						// Search next tu for this sequence
						fbSeqGetNextTU(
							Execute:= TRUE, 
							TU_Index:= TU_Index, 
							Destination:= TU_Table[TU_Index].Destination[1], 
							DestinationSlot:= TU_Table[TU_Index].DataSet.DestinationSlot, 
							Sequence:= TU_Table[TU_Index].DataSet.Sequence, 
							SubSequence:= TU_Table[TU_Index].DataSet.SubSequence, 
							Branch := Branch,
							BranchExclusionMode := BranchExclusionMode,
							TU_Table := TU_Table);

						State := 1;
					ELSE
						// Invalid TU data
						Busy := FALSE;
						State := 0;
					END_IF
				ELSE
					// No TU data, not part of a sequence
					Busy := FALSE;
					State := 0;	
				END_IF
			ELSE
				// No TU, stay
				Busy := FALSE;
				State := 0;
			END_IF
		END_IF
	
	// Search Next TU
	1:
		fbSeqGetNextTU(Execute:= FALSE, TU_Table := TU_Table);
		
		IF NOT fbSeqGetNextTU.Busy THEN
			IF NOT fbSeqGetNextTU.Error THEN
				NextTU_Index := fbSeqGetNextTU.NextTU_Index;
				// A next was found, store information to detect TU Data changes
				IF NextTU_Index > 0 THEN			
					M_AddToList(NextTU_Index, TU_Table[NextTU_Index]);
				END_IF
				
				Busy := FALSE;
				State := 0;
			ELSE
				// Error during search
				Error := TRUE;
				Busy := FALSE;
				State := 0;
			END_IF
		END_IF
ELSE
	// Default
	State := 0;
END_CASE

/// Add found data set to list
METHOD PRIVATE M_AddToList : BOOL
VAR_INPUT
	mTU_Index		: DINT;
END_VAR
VAR_IN_OUT
	mTU_Data		: ST_TU_Data;
END_VAR
VAR
	mIdx			: INT;
END_VAR
M_AddToList := FALSE;
		
FOR mIdx := 1 TO MAX_LIST_ENTRIES DO
	/// Check if already a slot is used for that destination
	IF NextTU_List[mIdx].Destination.eFunctionNumber = mTU_Data.Destination[1].eFunctionNumber AND
       NextTU_List[mIdx].Destination.ZoneNumber = mTU_Data.Destination[1].ZoneNumber AND
	   NextTU_List[mIdx].DestinationSlot = mTU_Data.DataSet.DestinationSlot THEN
	   
	    // Replace and store TU Data
	   	NextTU_List[mIdx].TU_Index := mTU_Index;
		NextTU_List[mIdx].Sequence := mTU_Data.DataSet.Sequence;
		NextTU_List[mIdx].SubSequence := mTU_Data.DataSet.SubSequence;
		NextTU_List[mIdx].Destination := mTU_Data.Destination[1];
		NextTU_List[mIdx].DestinationSlot := mTU_Data.DataSet.DestinationSlot;
		NextTU_List[mIdx].TU_ID_HashCode := mTU_Data.TU_ID.HashCode;
		NextTU_List[mIdx].TU_ID := mTU_Data.TU_ID.ASCII;
		NextTU_List[mIdx].AssignmentID := mTU_Data.AssignmentID;
	   	
		M_AddToList := TRUE;
	
	// If an empty slot is found
	ELSIF NextTU_List[mIdx].Destination.eFunctionNumber = E_FunctionNumber.F_BEGIN_FUNCTION THEN
		// Store TU Data
	   	NextTU_List[mIdx].TU_Index := mTU_Index;
		NextTU_List[mIdx].Sequence := mTU_Data.DataSet.Sequence;
		NextTU_List[mIdx].SubSequence := mTU_Data.DataSet.SubSequence;
		NextTU_List[mIdx].Destination := mTU_Data.Destination[1];
		NextTU_List[mIdx].DestinationSlot := mTU_Data.DataSet.DestinationSlot;
		NextTU_List[mIdx].TU_ID_HashCode := mTU_Data.TU_ID.HashCode;
		NextTU_List[mIdx].TU_ID := mTU_Data.TU_ID.ASCII;
		NextTU_List[mIdx].AssignmentID := mTU_Data.AssignmentID;
		
		M_AddToList := TRUE;
		
		ListCount := ListCount + 1;
	END_IF	
END_FOR
END_METHOD

/// Clears next TU list.
/// Returns true if succesful.
METHOD M_ClearList : BOOL
M_ClearList := MEMSET(ADR(NextTU_List), 0, SIZEOF(NextTU_List)) > 0;
END_METHOD

/// Checks if requesting TU is next in sequence
METHOD M_IsNextInSequence : BOOL // True = Next in Sequence, otherwise FALSE
VAR_INPUT
	mTU_Index		: DINT; // Requesting TU Index
END_VAR
VAR_IN_OUT
	mTU_Data		: ST_TU_Data; // Tu Data
END_VAR
VAR
	mIdx			: INT; // Iterator
END_VAR
M_IsNextInSequence := FALSE;
		
FOR mIdx := 1 TO ListCount DO
	// Check if an index is recorded as next
	IF mTU_Index = NextTU_List[mIdx].TU_Index THEN
		/// Ensure that recorded tu data entry is still the same as requesting Tu data
		IF mTU_Data.DataSet.Sequence = NextTU_List[mIdx].Sequence AND
		   mTU_Data.DataSet.SubSequence = NextTU_List[mIdx].SubSequence AND
		   mTU_Data.TU_ID.ASCII = NextTU_List[mIdx].TU_ID AND
		   mTU_Data.Destination[1].eFunctionNumber = NextTU_List[mIdx].Destination.eFunctionNumber AND
		   mTU_Data.Destination[1].ZoneNumber = NextTU_List[mIdx].Destination.ZoneNumber AND 
		   mTU_Data.DataSet.DestinationSlot = NextTU_List[mIdx].DestinationSlot THEN
		   
			M_IsNextInSequence := TRUE;
			RETURN;
		END_IF	
	END_IF
END_FOR
END_METHOD

END_FUNCTION_BLOCK

// ---- 20_Product/30_Toolbox/16_Sequencing/11_Strategies/FB_SeqEstimateNextTU.TcPOU
/// Estimates next awaiting TU after the requesting one of one specific destination.
FUNCTION_BLOCK FB_SeqEstimateNextTU IMPLEMENTS I_SeqEstimateNext
(************************************************************************************** 
* 	Application 		: BoxControl Framework 
* 	Revision 			: $Revision: 404877 $ 
* 	Revision date 		: $Date: 2018-04-26 14:10:34 +0200 (Thu, 26 Apr 2018) $ 
* 	Last changed by 	: $Author: b7ernsb $ 
* 	URL 				: $URL: http://almscdc.swisslog.com/repo/SWPD/Development/BoxControlFramework/21_Projects/BCF_2.0/trunk/BCF/BCF/JumpStart/20_Product/10_App/12_E_Functions/10_Lib/10_Conv/FB_FunctionConv.TcPOU $ 
* ------------------------------------------------------------------------------------ 
* 	© Swisslog AG 
* 	Swisslog is not liable for any usage of this source code that is not agreed 
* 	on between Swisslog and the other party. The mandatory legal liability remains 
* 	unaffected. 
* ------------------------------------------------------------------------------------ 
* 	Revision History: 
* 
* 	VERSION 		DATE 			INITIALS 			DESCRIPTION 
* 	0.1 			23.05.2018 		mbo 				Created.
*	0.2				31.10.2018		mbo					Race condition fixed for NextTUIndex
* 
**************************************************************************************)
VAR_INPUT
	Execute					: BOOL; // Requires rising edge for new request
	TU_Present				: BOOL; // A TU is present on branch A
	TU_Index				: DINT; // Waiting TU data index A
	Destination				: ST_PositionIdent; // Estimates next TU for this destination
	DestinationSlot			: INT; // Estimates next TU for this destination slot
	Branch					: I_BranchCheckpoint; // Branch to check for next branch
	BranchExclusionMode		: BOOL := FALSE; // False = TU on a branch is possible next, TRUE = TU on a branch is excluded as possible next
END_VAR
VAR_OUTPUT
	Busy					: BOOL; // Process ongoing
	Error					: BOOL; // Error during process (configuration error)
	NextTU_Index			: DINT; // Next expected TU of this sequence
END_VAR
VAR_IN_OUT
	TU_Table				: ARRAY[0..Conveyor.NUMBER_OF_TU_DATA] OF ST_TU_Data; // TU Table
END_VAR
VAR
	State					: INT; // State machine 0: Request 1: Search
	fbTrigExecute			: R_TRIG; // Trigger new request
	TU_DataChanged			: BOOL; // Data of stored NextTU have changed
	TU_LocationChanged		: BOOL; // Location of stored NextTU has changed
	TU_IsPartOfDestSequence : BOOL; // TU is part of the sequence to this destination
	SequenceDataPresent 	: BOOL; // Sequence data available
	NextAssignmentID		: UDINT; // Stored next assignment ID
	NextDestination			: ST_PositionIdent; // Stored destination information
	NextDestinationSlot		: INT; // Stored destination slot
	NextTU_ID				: STRING(Conveyor.TU_ID_STRINGLENGTH); // Stored next TU-ID HashCode
	NextSequence			: ULINT; // Stored next sequence
	NextSubSequence			: DINT; // Stored next sub sequence
	NextCheckpointID		: STRING(5); // Stored next checkpoint ID
	NextHaltSequencing		: BOOL; // Stored next halt sequencing bit
	fbSeqGetNextTU			: FB_SeqGetNextTU; // Get next following TU of this sequence
END_VAR

// Monitor new request trigger
fbTrigExecute(CLK := Execute);

CASE State OF
	// Wait for a new TU
	0:
		// Wait for new start trigger
		IF fbTrigExecute.Q THEN
			// Validate inputs
			IF Branch = 0 THEN
				Error := TRUE;
				RETURN;
			END_IF
			
			// Process started...
			Busy := TRUE;
			Error := FALSE;

			// When a requesting TU is present
			IF TU_Present THEN
				// If already a next TU was determined on a previous search, 
				// check if state or position has changed of it
				IF NextTU_Index > 0 THEN
					// Detect if the data of the monitored TU index has changed (e.g. TU data Add/Remove/Update)		
					TU_DataChanged := TU_Table[NextTU_Index].AssignmentID <> NextAssignmentID OR
									  TU_Table[NextTU_Index].TU_ID.ASCII <> NextTU_ID OR
									  TU_Table[NextTU_Index].DataSet.Sequence <> NextSequence OR
									  TU_Table[NextTU_Index].DataSet.SubSequence <> NextSubSequence OR
                                      TU_Table[NextTU_Index].Destination[1].eFunctionNumber <> NextDestination.eFunctionNumber OR
  									  TU_Table[NextTU_Index].Destination[1].ZoneNumber <> NextDestination.ZoneNumber OR
									  TU_Table[NextTU_Index].DataSet.DestinationSlot <> NextDestinationSlot OR
									  TU_Table[NextTU_Index].DataSet.HaltSequencing <> NextHaltSequencing;
			
					// Detect if the TU has changed the location (e.g. entered a new path)
					TU_LocationChanged := TU_Table[NextTU_Index].DataSet.CheckpointID <> NextCheckpointID;

					// Data changed, new release request		  
					IF TU_DataChanged OR TU_LocationChanged THEN
						M_ClearNextTU_Data();
					END_IF
				END_IF
					
				IF NextTU_Index > 0 THEN
					// No change of expected TU
					Busy := FALSE;
					State := 0;
				ELSIF TU_Index > 0 THEN
					// If the TU consists of sequencing information
					SequenceDataPresent := TU_Table[TU_Index].DataSet.Sequence > 0 AND
					                       TU_Table[TU_Index].Destination[1].eFunctionNumber > 0;
										   
					TU_IsPartOfDestSequence := TU_Table[TU_Index].Destination[1].eFunctionNumber = Destination.eFunctionNumber AND
					 						   TU_Table[TU_Index].Destination[1].ZoneNumber = Destination.ZoneNumber AND
											   TU_Table[TU_Index].DataSet.DestinationSlot = DestinationSlot;
					
					IF SequenceDataPresent AND TU_IsPartOfDestSequence THEN
						fbSeqGetNextTU(
							Execute:= TRUE, 
							TU_Index:= TU_Index, 
							Destination:= TU_Table[TU_Index].Destination[1], 
							DestinationSlot:= TU_Table[TU_Index].DataSet.DestinationSlot, 
							Sequence:= TU_Table[TU_Index].DataSet.Sequence, 
							SubSequence:= TU_Table[TU_Index].DataSet.SubSequence, 
							Branch := Branch,
							BranchExclusionMode := BranchExclusionMode,
							TU_Table := TU_Table);
							
						State := 1;
					ELSE
						// Invalid TU data
						Busy := FALSE;
						State := 0;
					END_IF
				ELSE
					// No TU data, not part of a sequence
					Busy := FALSE;
					State := 0;	
				END_IF
			ELSE
				// No TU, stay
				Busy := FALSE;
				State := 0;
			END_IF
		END_IF
	
	// Search Next TU
	1:
		fbSeqGetNextTU(
			Execute:= FALSE, 
			TU_Index:= TU_Index, 
			Destination:= TU_Table[TU_Index].Destination[1], 
			DestinationSlot:= TU_Table[TU_Index].DataSet.DestinationSlot, 
			Sequence:= TU_Table[TU_Index].DataSet.Sequence, 
			SubSequence:= TU_Table[TU_Index].DataSet.SubSequence, 
			Branch := Branch,
			BranchExclusionMode := BranchExclusionMode,
			NextTU_Index => NextTU_Index,
			TU_Table := TU_Table);
		
		IF NOT fbSeqGetNextTU.Busy THEN
			IF NOT fbSeqGetNextTU.Error THEN
				// A next was found, store information to detect TU Data changes
				IF NextTU_Index > 0 THEN
					NextAssignmentID := TU_Table[NextTU_Index].AssignmentID; 
					NextTU_ID := TU_Table[NextTU_Index].TU_ID.ASCII;
					NextSequence := TU_Table[NextTU_Index].DataSet.Sequence;
					NextSubSequence	:= TU_Table[NextTU_Index].DataSet.SubSequence;
					NextCheckpointID := TU_Table[NextTU_Index].DataSet.CheckpointID;
					NextDestination := TU_Table[NextTU_Index].Destination[1];
					NextDestinationSlot := TU_Table[NextTU_Index].DataSet.DestinationSlot;
					NextHaltSequencing := TU_Table[NextTU_Index].DataSet.HaltSequencing;

				// No next found for this specific destination
				ELSE
					M_ClearNextTU_Data();
				END_IF
				
				Busy := FALSE;
				State := 0;
			ELSE
				// Error during search
				Error := TRUE;
				Busy := FALSE;
				State := 0;
			END_IF
		END_IF
ELSE
	// Default
	State := 0;
END_CASE

/// Reset next expected TU, so on a new request a new search is triggered
METHOD M_ResetExpectedTU 
VAR_INPUT
END_VAR
NextTU_Index := 0;
END_METHOD

/// Clears next tu data
METHOD PROTECTED M_ClearNextTU_Data
VAR_INPUT
END_VAR
NextTU_Index := 0;
NextAssignmentID := 0; 
NextTU_ID := '';
NextSequence := 0;
NextSubSequence	:= 0;
NextCheckpointID := '';
NextDestination.eFunctionNumber := 0;
NextDestination.ZoneNumber := 0;
NextDestinationSlot := 0;
NextHaltSequencing :=  FALSE;
END_METHOD

/// Checks if requesting TU is next in sequence
METHOD M_IsNextInSequence : BOOL // True = Next in Sequence, otherwise FALSE
VAR_INPUT
	mTU_Index		: DINT; // Requesting TU Index
END_VAR
VAR_IN_OUT
	mTU_Data			: ST_TU_Data; // Tu Data
END_VAR

IF NextTU_Index > 0 THEN
	// Check whether the requesting TU is the same, as the next sequence TU was stored
	IF TU_Index = NextTU_Index AND
	   mTU_Data.DataSet.Sequence = NextSequence AND
	   mTU_Data.DataSet.SubSequence = NextSubSequence AND
	   mTU_Data.TU_ID.ASCII = NextTU_ID AND
	   mTU_Data.DataSet.CheckpointID = NextCheckpointID AND
	   mTU_Data.Destination[1].eFunctionNumber = NextDestination.eFunctionNumber AND
	   mTU_Data.Destination[1].ZoneNumber = NextDestination.ZoneNumber AND 
	   mTU_Data.DataSet.DestinationSlot = NextDestinationSlot THEN
	   
	   	// Release
		M_IsNextInSequence := TRUE;
	ELSE
	   M_IsNextInSequence := FALSE;
	END_IF
ELSE
	M_IsNextInSequence := FALSE;
END_IF
END_METHOD

END_FUNCTION_BLOCK

// ---- 20_Product/30_Toolbox/16_Sequencing/11_Strategies/FB_SeqEstimateStreamRange.TcPOU
/// Estimates all next awaiting TUs of one specific destination stream considering 
/// the configured branch.
FUNCTION_BLOCK FB_SeqEstimateStreamRange 
(************************************************************************************** 
* 	Application 		: BoxControl Framework 
* 	Revision 			: $Revision: 404877 $ 
* 	Revision date 		: $Date: 2018-04-26 14:10:34 +0200 (Thu, 26 Apr 2018) $ 
* 	Last changed by 	: $Author: b7ernsb $ 
* 	URL 				: $URL: http://almscdc.swisslog.com/repo/SWPD/Development/BoxControlFramework/21_Projects/BCF_2.0/trunk/BCF/BCF/JumpStart/20_Product/10_App/12_E_Functions/10_Lib/10_Conv/FB_FunctionConv.TcPOU $ 
* ------------------------------------------------------------------------------------ 
* 	© Swisslog AG 
* 	Swisslog is not liable for any usage of this source code that is not agreed 
* 	on between Swisslog and the other party. The mandatory legal liability remains 
* 	unaffected. 
* ------------------------------------------------------------------------------------ 
* 	Revision History: 
* 
* 	VERSION 		DATE 			INITIALS 			DESCRIPTION 
* 	0.1 			23.05.2018 		mbo 				Created.
*	0.2				08.02.2019		mbo					Renamed + Racecondition
* 
**************************************************************************************)
VAR_INPUT
	Execute					: BOOL; // Requires rising edge for new request
	TU_Present				: BOOL; // A TU is present on branch A
	TU_Index				: DINT; // Waiting TU data index A
	Destination				: ST_PositionIdent; // Estimates next TU for this destination
	DestinationSlot			: INT; // Estimates next TU for this destination slot
	Branch					: I_BranchCheckpoint; // Branch to check for next branch
	BranchExclusionMode		: BOOL := FALSE; // False = TU on a branch is possible next, TRUE = TU on a branch is excluded as possible next
	RangeLimit				: INT; // Specifies how many entries of the list serve as valid. (0=All available)
END_VAR
VAR_OUTPUT
	Busy					: BOOL; // Process ongoing
	Error					: BOOL; // Error during process (configuration error)
	NextTU_Index			: DINT; // Next expected TU of this sequence
END_VAR
VAR_IN_OUT
	TU_Table				: ARRAY[0..Conveyor.NUMBER_OF_TU_DATA] OF ST_TU_Data; // TU Table
END_VAR
VAR
	State					: INT; // State machine 0: Request 1: Search
	fbTrigExecute			: R_TRIG; // Trigger new request
	TU_DataChanged			: BOOL; // Data of stored NextTU have changed
	TU_LocationChanged		: BOOL; // Location of stored NextTU has changed
	TU_IsPartOfDestSequence : BOOL; // TU is part of the sequence to this destination
	SequenceDataPresent 	: BOOL; // Sequence data available
	NextAssignmentID		: UDINT; // Stored next assignment ID
	NextDestination			: ST_PositionIdent; // Stored destination information
	NextDestinationSlot		: INT; // Stored destination slot
	NextTU_ID				: STRING(Conveyor.TU_ID_STRINGLENGTH); // Stored next TU-ID HashCode
	NextSequence			: ULINT; // Stored next sequence
	NextSubSequence			: DINT; // Stored next sub sequence
	NextCheckpointID		: STRING(5); // Stored next checkpoint ID
	NextHaltSequencing		: BOOL; // Stored next halt sequencing bit
	fbSeqBuildStream		: FB_SeqBuildStream; // Instance to build range of stream
END_VAR

// Monitor new request trigger
fbTrigExecute(CLK := Execute);

CASE State OF
	// Wait for a new TU
	0:
		// Wait for new start trigger
		IF fbTrigExecute.Q THEN
			// Validate inputs
			IF Branch = 0 THEN
				Error := TRUE;
				RETURN;
			END_IF
			
			// Process started...
			Busy := TRUE;
			Error := FALSE;

			// When a requesting TU is present
			IF TU_Present THEN
				// If already a next TU was determined on a previous search, 
				// check if state or position has changed of it
				IF NextTU_Index > 0 THEN
					// Detect if the data of the monitored TU index has changed (e.g. TU data Add/Remove/Update)		
					TU_DataChanged := TU_Table[NextTU_Index].AssignmentID <> NextAssignmentID OR
									  TU_Table[NextTU_Index].TU_ID.ASCII <> NextTU_ID OR
									  TU_Table[NextTU_Index].DataSet.Sequence <> NextSequence OR
									  TU_Table[NextTU_Index].DataSet.SubSequence <> NextSubSequence OR
                                      TU_Table[NextTU_Index].Destination[1].eFunctionNumber <> NextDestination.eFunctionNumber OR
  									  TU_Table[NextTU_Index].Destination[1].ZoneNumber <> NextDestination.ZoneNumber OR
									  TU_Table[NextTU_Index].DataSet.DestinationSlot <> NextDestinationSlot OR
									  TU_Table[NextTU_Index].DataSet.HaltSequencing <> NextHaltSequencing;
			
					// Detect if the TU has changed the location (e.g. entered a new path)
					TU_LocationChanged := TU_Table[NextTU_Index].DataSet.CheckpointID <> NextCheckpointID;

					// Data changed, new release request		  
					IF TU_DataChanged OR TU_LocationChanged THEN
						M_ClearNextTU_Data();
					END_IF
				END_IF
					
				IF NextTU_Index > 0 THEN
					// No change of expected TU
					Busy := FALSE;
					State := 0;
				ELSIF TU_Index > 0 THEN
					// If the TU consists of sequencing information
					SequenceDataPresent := TU_Table[TU_Index].DataSet.Sequence > 0 AND
					                       TU_Table[TU_Index].Destination[1].eFunctionNumber > 0;
										   
					TU_IsPartOfDestSequence := TU_Table[TU_Index].Destination[1].eFunctionNumber = Destination.eFunctionNumber AND
					 						   TU_Table[TU_Index].Destination[1].ZoneNumber = Destination.ZoneNumber AND
											   TU_Table[TU_Index].DataSet.DestinationSlot = DestinationSlot;
					
					IF SequenceDataPresent AND TU_IsPartOfDestSequence THEN
						
						fbSeqBuildStream(
							Execute:= TRUE,
							Destination:= TU_Table[TU_Index].Destination[1], 
							DestinationSlot:= TU_Table[TU_Index].DataSet.DestinationSlot, 
							Branch := Branch,
							BranchExclusionMode := BranchExclusionMode,
							TU_Table := TU_Table);
							
						State := 1;
					ELSE
						// Invalid TU data
						Busy := FALSE;
						State := 0;
					END_IF
				ELSE
					// No TU data, not part of a sequence
					Busy := FALSE;
					State := 0;	
				END_IF
			ELSE
				// No TU, stay
				Busy := FALSE;
				State := 0;
			END_IF
		END_IF
	
	// Search Next TU
	1:
		fbSeqBuildStream(
			Execute:= FALSE,
			Destination:= TU_Table[TU_Index].Destination[1], 
			DestinationSlot:= TU_Table[TU_Index].DataSet.DestinationSlot, 
			Branch := Branch,
			BranchExclusionMode := BranchExclusionMode,
			NextTU_Index => NextTU_Index,
			TU_Table := TU_Table);
		
		IF NOT fbSeqBuildStream.Busy THEN
			IF NOT fbSeqBuildStream.Error THEN
				// A next was found, store information to detect TU Data changes
				IF NextTU_Index > 0 THEN
					NextAssignmentID := TU_Table[NextTU_Index].AssignmentID; 
					NextTU_ID := TU_Table[NextTU_Index].TU_ID.ASCII;
					NextSequence := TU_Table[NextTU_Index].DataSet.Sequence;
					NextSubSequence	:= TU_Table[NextTU_Index].DataSet.SubSequence;
					NextCheckpointID := TU_Table[NextTU_Index].DataSet.CheckpointID;
					NextDestination := TU_Table[NextTU_Index].Destination[1];
					NextDestinationSlot := TU_Table[NextTU_Index].DataSet.DestinationSlot;
					NextHaltSequencing := TU_Table[NextTU_Index].DataSet.HaltSequencing;
					
				// No next found for this specific destination
				ELSE
					M_ClearNextTU_Data();
				END_IF
				
				Busy := FALSE;
				State := 0;
			ELSE
				// Error during search
				Error := TRUE;
				Busy := FALSE;
				State := 0;
			END_IF
		END_IF
ELSE
	// Default
	State := 0;
END_CASE

/// Reset next expected TU, so on a new request a new search is triggered
METHOD M_ResetExpectedTU 
VAR_INPUT
END_VAR
NextTU_Index := 0;
END_METHOD

/// Checks if requesting TU is next in sequence
METHOD M_IsNextInSequence : BOOL // True = Next in Sequence, otherwise FALSE
VAR_INPUT
	mTU_Index		: DINT; // Requesting TU Index
END_VAR
VAR_IN_OUT
	mTU_Data			: ST_TU_Data; // Tu Data
END_VAR

IF NextTU_Index > 0 THEN
	M_IsNextInSequence := fbSeqBuildStream.M_IsTU_OnStream(
												mRangeLimit := RangeLimit,
												mTU_Index := TU_Index,
												mTU_Data := mTU_Data);
ELSE
	M_IsNextInSequence := FALSE;
END_IF
END_METHOD

/// Clears next tu data
METHOD PROTECTED M_ClearNextTU_Data
VAR_INPUT
END_VAR
NextTU_Index := 0;
NextAssignmentID := 0; 
NextTU_ID := '';
NextSequence := 0;
NextSubSequence	:= 0;
NextCheckpointID := '';
NextDestination.eFunctionNumber := 0;
NextDestination.ZoneNumber := 0;
NextDestinationSlot := 0;
END_METHOD

END_FUNCTION_BLOCK

// ---- 20_Product/30_Toolbox/16_Sequencing/11_Strategies/FB_SeqMerge2W.TcPOU
/// Sequence strategy Merge 2-Way
/// This strategy is able to ensure sequencing from two branches.
/// Remark: Decision can take multiple cycles, check busy and reset FB before new request.
/// Uses recursive calls - User has to ensure to not generate a loop (Tested up to 350 jumps)
FUNCTION_BLOCK FB_SeqMerge2W IMPLEMENTS I_BranchCheckpoint
(************************************************************************************** 
* 	Application 		: BoxControl Framework 
* 	Revision 			: $Revision: 404877 $ 
* 	Revision date 		: $Date: 2018-04-26 14:10:34 +0200 (Thu, 26 Apr 2018) $ 
* 	Last changed by 	: $Author: b7ernsb $ 
* 	URL 				: $URL: http://almscdc.swisslog.com/repo/SWPD/Development/BoxControlFramework/21_Projects/BCF_2.0/trunk/BCF/BCF/JumpStart/20_Product/10_App/12_E_Functions/10_Lib/10_Conv/FB_FunctionConv.TcPOU $ 
* ------------------------------------------------------------------------------------ 
* 	© Swisslog AG 
* 	Swisslog is not liable for any usage of this source code that is not agreed 
* 	on between Swisslog and the other party. The mandatory legal liability remains 
* 	unaffected. 
* ------------------------------------------------------------------------------------ 
* 	Revision History: 
* 
* 	VERSION 		DATE 			INITIALS 			DESCRIPTION 
* 	0.1 			01.05.2018 		mbo 				Created.
* 
**************************************************************************************)
VAR_INPUT
	Execute					: BOOL; // Requires rising edge for new request
	CheckpointID			: STRING(5); // Checkpoint ID, used to identify location of TUs
	TU_PresentA				: BOOL; // A TU is present on branch A
	TU_IndexA				: DINT; // Waiting TU data index A
	TU_PresentB 			: BOOL; // A TU is present on branch B
	TU_IndexB				: DINT; // Waiting TU data index B
	iBranchA				: I_BranchCheckpoint; // Previous decision point on this branch
	iBranchB				: I_BranchCheckpoint; // Previous decision point on this branch
	iEstimateNextServiceA	: I_SeqEstimateNext; // Service to estimate possible next in order to save calculation time (optional)
	iEstimateNextServiceB	: I_SeqEstimateNext; // Service to estimate possible next in order to save calculation time (optional)
	EnableWarningA			: BOOL; // When enabled, warning is active if a TU is waiting, RisingEdge restarts Timer
	EnableWarningB			: BOOL; // When enabled, warning is active if a TU is waiting, RisingEdge restarts Timer
END_VAR

VAR_IN_OUT 
	TU_Table				: ARRAY[0..Conveyor.NUMBER_OF_TU_DATA] OF ST_TU_Data; // TU Table
END_VAR

VAR_OUTPUT
	Busy					: BOOL; // Process ongoing
	Error					: BOOL; // Error during process
	ReleaseA				: BOOL; // Release TU on branch A
	ReleaseB				: BOOL; // Release TU on branch B
	TimeoutWaitA			: BOOL; // Warning, TU is waiting longer than P_WarningTime
	TimeoutWaitB			: BOOL; // Warning, TU is waiting longer than P_WarningTime
END_VAR

VAR
	fbBranchA				: FB_SeqBranch; // Branch A 
	fbBranchB				: FB_SeqBranch; // Branch B
	UpdateCheckpointID		: BOOL; // Enable update ceckpoint IDs of waiting Tus
	WarningTime				: TIME := SequencingParameter.DEFAULT_WARNING_TIME; // Time after a warning gets reported.
	fbWarnA					: TON; // Timer warning A
	fbWarnB					: TON; // Timer warning B
END_VAR

// Check inputs
IF TU_IndexA < 0 OR TU_IndexB < 0 THEN
	Error := TRUE;
	RETURN;
END_IF

// Initialize values
Error := FALSE;

// If branch A is configured, update waiting TU with Checkpoint ID
IF iBranchA <> 0 AND UpdateCheckpointID THEN
	F_UpdateCheckpointID(
		Enable := TU_PresentA AND TU_IndexA > 0,
		CheckpointID := iBranchA.P_CheckpointID,
		TU_Data := TU_Table[TU_IndexA]);
END_IF

// If branch B is configured, update waiting TU with Checkpoint ID
IF iBranchB <> 0 AND UpdateCheckpointID THEN
	F_UpdateCheckpointID(
		Enable := TU_PresentB AND TU_IndexB > 0,
		CheckpointID := iBranchB.P_CheckpointID,
		TU_Data := TU_Table[TU_IndexB]);	
END_IF

fbBranchA(
	Execute:= Execute, 
	TU_Present:= TU_PresentA, 
	TU_Index:= TU_IndexA, 
	Branch:= iBranchA, 
	iEstimateNextService:= iEstimateNextServiceA, 
	Release=> ReleaseA, 
	TU_Table:= TU_Table);
	
fbBranchB(
	Execute:= Execute, 
	TU_Present:= TU_PresentB, 
	TU_Index:= TU_IndexB, 
	Branch:= iBranchB, 
	iEstimateNextService:= iEstimateNextServiceB, 
	Release=> ReleaseB, 
	TU_Table:= TU_Table);
	
Busy := fbBranchA.Busy OR fbBranchB.Busy;
Error := fbBranchA.Error OR fbBranchB.Error;

fbWarnA(IN := EnableWarningA AND TU_PresentA, PT := WarningTime);
fbWarnB(IN := EnableWarningB AND TU_PresentB, PT := WarningTime);

TimeoutWaitA := fbWarnA.Q;
TimeoutWaitB := fbWarnB.Q;

/// Searches if a checkpoint can be found on a specific branch
/// Returns true if found, false = not found
METHOD M_IsOnBranches : BOOL
VAR_INPUT
	mRecursive	: BOOL := FALSE; // Search recursive through the whole tree
END_VAR
VAR_IN_OUT CONSTANT
	// Last checkpoint id	
	mCheckpointID	: STRING(5);
END_VAR

IF mCheckpointID = '' THEN
	M_IsOnBranches := FALSE;
	RETURN;
END_IF

IF mCheckpointID = P_CheckpointID THEN
	M_IsOnBranches := TRUE;
	RETURN;
END_IF

// When its requested that its branches are checked as well
IF mRecursive THEN
	IF iBranchA <> 0 THEN
		 IF iBranchA.M_IsOnBranches(TRUE, mCheckpointId) THEN;
			M_IsOnBranches := TRUE;
			RETURN;
		END_IF
	END_IF
	
	IF iBranchB <> 0 THEN
		IF iBranchB.M_IsOnBranches(TRUE, mCheckpointId) THEN;
			M_IsOnBranches := TRUE;
			RETURN;
		END_IF
	END_IF
END_IF
END_METHOD

METHOD M_Reset : BOOL
VAR_INPUT
END_VAR
fbBranchA.M_Reset();
fbBranchB.M_Reset();
END_METHOD

/// Identifier for checkpoint
{attribute 'monitoring' := 'call'}
{attribute 'suppress_wrn_C0410'}
PROPERTY P_CheckpointID : REFERENCE TO STRING(5)
GET
P_CheckpointID REF= CheckpointID;
END_GET
END_PROPERTY

/// TU Entries scanned per cycle
PROPERTY P_EntriesPerCycle : DINT // Default 600
GET
P_EntriesPerCycle := fbBranchA.P_EntriesPerCycle;
END_GET
SET
fbBranchA.P_EntriesPerCycle := P_EntriesPerCycle;
fbBranchB.P_EntriesPerCycle := P_EntriesPerCycle;
END_SET
END_PROPERTY

/// When enabled, Checkpoint ID of waiting TUs is updated automatically with previous Branch ID
PROPERTY P_UpdateCheckpointID : BOOL
GET
P_UpdateCheckpointID := UpdateCheckpointID;
END_GET
SET
UpdateCheckpointID := P_UpdateCheckpointID;
END_SET
END_PROPERTY

/// Time after Warning gets reported
PROPERTY P_WarningTime : TIME
GET
P_WarningTime := WarningTime;
END_GET
SET
WarningTime := P_WarningTime;
END_SET
END_PROPERTY

END_FUNCTION_BLOCK

// ---- 20_Product/30_Toolbox/16_Sequencing/12_Helper/FB_SeqConveyorLane.TcPOU
// Object representing a conveyor lane consisting of multiple zones
FUNCTION_BLOCK FB_SeqConveyorLane
(************************************************************************************** 
* 	Application 		: BoxControl Framework 
* 	Revision 			: $Revision: 404877 $ 
* 	Revision date 		: $Date: 2018-04-26 14:10:34 +0200 (Thu, 26 Apr 2018) $ 
* 	Last changed by 	: $Author: b7ernsb $ 
* 	URL 				: $URL: http://almscdc.swisslog.com/repo/SWPD/Development/BoxControlFramework/21_Projects/BCF_2.0/trunk/BCF/BCF/JumpStart/20_Product/10_App/12_E_Functions/10_Lib/10_Conv/FB_FunctionConv.TcPOU $ 
* ------------------------------------------------------------------------------------ 
* 	© Swisslog AG 
* 	Swisslog is not liable for any usage of this source code that is not agreed 
* 	on between Swisslog and the other party. The mandatory legal liability remains 
* 	unaffected. 
* ------------------------------------------------------------------------------------ 
* 	Revision History: 
* 
* 	VERSION 		DATE 			INITIALS 			DESCRIPTION 
* 	0.1 			06.05.2019 		ber 				Created.

* 
**************************************************************************************)
VAR_INPUT
	Positions						: ARRAY [1..MAX_LANE_SIZE] OF ST_PositionIdent; // Index 1: Outfeed position of the lane 
END_VAR
VAR
	PositionCount					: DINT; // Amount of positions in the lane
	OnlySequencingTU				: BOOL:= TRUE; // Only allow TU with sequencing data to enter the lane
	Idx								: DINT;
END_VAR

VAR CONSTANT
	MAX_LANE_SIZE					: DINT:=SequencingParameter.MAX_LANE_SIZE; // Maximal number of zones in a conveyor lane
END_VAR

PositionCount:= 0;	
// Determine amount of positions in the lane
FOR Idx:=1 TO MAX_LANE_SIZE DO
	IF Positions[Idx].eFunctionNumber>0 THEN
		PositionCount:= PositionCount+1;
	END_IF
END_FOR

/// Returns all TU indices currently present in the lane
METHOD M_GetAllTU : BOOL // True = execution sucessfull, else false
VAR_IN_OUT
	mTU_Indices	: ARRAY [*] OF DINT; // List of all TU data indices in the lane
END_VAR
VAR
	mIdx		: DINT;
	mTU_Index	: DINT;
	mCount		: DINT;
END_VAR
MEMSET(ADR(mTU_Indices^), 0,  DINT_TO_UDINT((UPPER_BOUND(mTU_Indices,1)- LOWER_BOUND(mTU_Indices,1)+1)*SIZEOF(mTU_Indices^)));	
mCount:= LOWER_BOUND(mTU_Indices,1);
M_GetAllTU:= TRUE;	

// Loop through lane
FOR mIdx:=1 TO PositionCount DO	
	
	mTU_Index:= F_GetTU_DataIndex(Positions[mIdx].eFunctionNumber, Positions[mIdx].ZoneNumber);
	
	// If a TU index is present on the zone	
	IF mTU_Index > 0 THEN

		// Input array has enough space
		IF mCount <= UPPER_BOUND( mTU_Indices,1) THEN
			
			mTU_Indices[mCount]:= mTU_Index;
			mCount:= mCount+1;
		
		ELSE // Input array too small
	
			MEMSET(ADR(mTU_Indices^), 0, DINT_TO_UDINT((UPPER_BOUND(mTU_Indices,1)- LOWER_BOUND(mTU_Indices,1)+1)*SIZEOF(mTU_Indices^)));		
			M_GetAllTU:= FALSE;	
			EXIT;		
		END_IF

	END_IF
END_FOR
END_METHOD

// Get TU Index on first occupied position (nearest to the infeed)
METHOD M_GetFirstTU : DINT // TU index
VAR
	mIdx				: DINT;
END_VAR
VAR_INST
	TransportCtrlData	: ST_TransportControlData;	
END_VAR
M_GetFirstTU:=0;

// Loop through lane from infeed to outfeed
FOR mIdx:=0 TO PositionCount-1 DO	
	
	TransportCtrlData:= F_GetTransportControlData(Positions[PositionCount-mIdx].eFunctionNumber, Positions[PositionCount-mIdx].ZoneNumber);

	// Finish search when a TU was found	
	IF  TransportCtrlData.NumberOfPresentTUs > 0 THEN
		M_GetFirstTU:=F_GetTU_DataIndex( Positions[PositionCount-mIdx].eFunctionNumber, Positions[PositionCount-mIdx].ZoneNumber);
		EXIT;
	END_IF
	
END_FOR
END_METHOD

// Get TU Index on last occupied position (nearest to the outfeed)
METHOD M_GetLastTU : DINT // TU index
VAR
	mIdx				: DINT;
END_VAR
VAR_INST
	TransportCtrlData	: ST_TransportControlData;	
END_VAR
M_GetLastTU:=0;

// Loop through lane from outfeed to infeed
FOR mIdx:=1 TO PositionCount DO	
	
	TransportCtrlData:= F_GetTransportControlData(Positions[mIdx].eFunctionNumber, Positions[mIdx].ZoneNumber);
	
	// Finish search when a TU was found
	IF  TransportCtrlData.NumberOfPresentTUs > 0 THEN
		M_GetLastTU:= F_GetTU_DataIndex( Positions[mIdx].eFunctionNumber, Positions[mIdx].ZoneNumber);
		EXIT;
	END_IF
	
END_FOR
END_METHOD

// Returns number of empty zones in the lane
METHOD M_GetNrOfEmptyZones : DINT 
VAR
	mIdx				: DINT;
	mEmptyPosition_Count: DINT;
END_VAR
VAR_INST
	TransportCtrlData	: ST_TransportControlData;	
END_VAR
// Loop through lane from outfeed to infeed
FOR mIdx:=1 TO PositionCount DO	
	
	TransportCtrlData:= F_GetTransportControlData(Positions[mIdx].eFunctionNumber, Positions[mIdx].ZoneNumber);
	
	// Increase count when no TU is present on the zone
	IF  TransportCtrlData.NumberOfPresentTUs = 0 THEN
		mEmptyPosition_Count:=mEmptyPosition_Count+1;
	END_IF
	
END_FOR

M_GetNrOfEmptyZones:= mEmptyPosition_Count;
END_METHOD

// Returns number of occupied zones in the lane
METHOD M_GetNrOfOccupiedZones : DINT 
VAR
	mIdx				: DINT;
	mTU_Count			: DINT;
END_VAR
VAR_INST
	TransportCtrlData	: ST_TransportControlData;	
END_VAR
// Loop through lane from outfeed to infeed
FOR mIdx:=1 TO PositionCount DO	
	
	TransportCtrlData:= F_GetTransportControlData(Positions[mIdx].eFunctionNumber, Positions[mIdx].ZoneNumber);

	// Increase count when TU is present on the zone	
	IF  TransportCtrlData.NumberOfPresentTUs > 0 THEN
		mTU_Count:=mTU_Count+1;
	END_IF
	
END_FOR

M_GetNrOfOccupiedZones:= mTU_Count;
END_METHOD

/// Returns all TU indices (which have sequencing data)  after the last sequence error (sequence error nearest to the lane outfeed)
METHOD M_GetTUs_AfterLastError : BOOL; // True = execution successfull, else false
VAR_IN_OUT
	mTU_Indices					: ARRAY [*] OF DINT; // List of TU data indices after the error
	mTU_Table					: ARRAY[0..Conveyor.NUMBER_OF_TU_DATA] OF ST_TU_Data; // TU Table
END_VAR
VAR 
	mIdx						: DINT;
	mTU_IdxTemp					: DINT;
	mTU_IdxOutput				: DINT; 
	mCount						: DINT;
	mSequenceErrorFound			: BOOL;
END_VAR
VAR_INST
	TransportCtrlDataOutput		: ST_TransportControlData; 
	TransportCtrlDataTemp		: ST_TransportControlData; 
END_VAR
MEMSET(ADR(mTU_Indices^), 0, DINT_TO_UDINT((UPPER_BOUND(mTU_Indices,1)- LOWER_BOUND(mTU_Indices,1)+1)*SIZEOF(mTU_Indices^)));		
M_GetTUs_AfterLastError:=TRUE;
mCount:= LOWER_BOUND(mTU_Indices,1);

// Loop through lane
FOR mIdx:=1 TO PositionCount DO
	
	TransportCtrlDataTemp:= F_GetTransportControlData(Positions[mIdx].eFunctionNumber, Positions[mIdx].ZoneNumber);
	mTU_IdxTemp:= F_GetTU_DataIndex(Positions[mIdx].eFunctionNumber, Positions[mIdx].ZoneNumber);

	// Check if there is TU with sequencing information	
	IF  TransportCtrlDataTemp.NumberOfPresentTUs > 0 AND mTU_Table[mTU_IdxTemp].DataSet.Sequence > 0 THEN
		
		// New TU  with sequencing data found		
		IF mTU_IdxOutput = 0 THEN
			
			// Set TU as comparable
			mTU_IdxOutput := mTU_IdxTemp;
			TransportCtrlDataOutput:= TransportCtrlDataTemp;
		
		// Check if both TUs have the same destination ( belong to the same stream).	
		ELSIF  mTU_Table[mTU_IdxOutput].Destination[1].eFunctionNumber <> mTU_Table[mTU_IdxTemp].Destination[1].eFunctionNumber OR
				mTU_Table[mTU_IdxOutput].Destination[1].ZoneNumber <> mTU_Table[mTU_IdxTemp].Destination[1].ZoneNumber OR
				mTU_Table[mTU_IdxOutput].DataSet.DestinationSlot <> mTU_Table[mTU_IdxTemp].DataSet.DestinationSlot THEN
		
			// TUs dont belong to the same stream!!
			M_GetTUs_AfterLastError:=FALSE;
			EXIT;	
				
		
		ELSE // Compare with TU nearer to the output		
		
			// Check if TU which is nearer to the output is located higher in the stream	
			IF	mTU_Table[mTU_IdxOutput].DataSet.Sequence >  mTU_Table[mTU_IdxTemp].DataSet.Sequence OR 
				(mTU_Table[mTU_IdxOutput].DataSet.Sequence =  mTU_Table[mTU_IdxTemp].DataSet.Sequence AND
				mTU_Table[mTU_IdxOutput].DataSet.SubSequence >  mTU_Table[mTU_IdxTemp].DataSet.SubSequence)THEN				
				
				// Sequence error detected
				mSequenceErrorFound:= TRUE;
				EXIT;
				
			ELSE // TUs are in correct sequencing order
	
				// Set TU as new comparable
				mTU_IdxOutput := mTU_IdxTemp;
				TransportCtrlDataOutput:= TransportCtrlDataTemp;			
			END_IF	
		END_IF
		
		// If input list is big enough, add the found index
		IF  mCount <= UPPER_BOUND(mTU_Indices,1) THEN
				
			// Add index to list
			mTU_Indices[mCount]:= mTU_IdxTemp;
			mCount:= mCount+1;
				
		ELSE // Array too small
			M_GetTUs_AfterLastError:=FALSE;
			EXIT;
		END_IF
		
	END_IF
END_FOR


IF NOT mSequenceErrorFound OR NOT M_GetTUs_AfterLastError THEN
	MEMSET(ADR(mTU_Indices^), 0, DINT_TO_UDINT((UPPER_BOUND(mTU_Indices,1)- LOWER_BOUND(mTU_Indices,1)+1)*SIZEOF(mTU_Indices^)));		
END_IF
END_METHOD

/// Checks if there is a sequence error pending  within the lane
METHOD M_HasSquenceError : BOOL // True = sequence error pending, else false
VAR_IN_OUT
	mTU_Table					: ARRAY[0..Conveyor.NUMBER_OF_TU_DATA] OF ST_TU_Data; // TU Data Table
END_VAR
VAR 
	mTU_IdxTemp					: DINT;
	mTU_IdxOutput				: DINT; 
	mIdx						: DINT;
	mSequenceErrorFound			: BOOL;
END_VAR
VAR_INST
	TransportCtrlDataOutput		: ST_TransportControlData; 
	TransportCtrlDataTemp		: ST_TransportControlData;
END_VAR
mSequenceErrorFound:=FALSE;

// Loop through lane from outfeed to infeed
FOR mIdx:=1 TO PositionCount DO
	
	TransportCtrlDataTemp:= F_GetTransportControlData(Positions[mIdx].eFunctionNumber, Positions[mIdx].ZoneNumber);
	mTU_IdxTemp:= F_GetTU_DataIndex(Positions[mIdx].eFunctionNumber, Positions[mIdx].ZoneNumber);

	// Check if there is TU with sequencing information	
	IF  TransportCtrlDataTemp.NumberOfPresentTUs > 0 AND mTU_Table[mTU_IdxTemp].DataSet.Sequence > 0 THEN
		
		// New TU  with sequencing data found		
		IF mTU_IdxOutput = 0 THEN
			
			// Set TU as comparable
			mTU_IdxOutput := mTU_IdxTemp;
			TransportCtrlDataOutput:= TransportCtrlDataTemp;
		
		// Check if both TUs have the same destination ( belong to the same stream).	
		ELSIF  mTU_Table[mTU_IdxOutput].Destination[1].eFunctionNumber <> mTU_Table[mTU_IdxTemp].Destination[1].eFunctionNumber OR
				mTU_Table[mTU_IdxOutput].Destination[1].ZoneNumber <> mTU_Table[mTU_IdxTemp].Destination[1].ZoneNumber OR
				mTU_Table[mTU_IdxOutput].DataSet.DestinationSlot <> mTU_Table[mTU_IdxTemp].DataSet.DestinationSlot THEN
		

			mSequenceErrorFound:=TRUE;
			EXIT;	
				
		
		ELSE // Compare with TU nearer to the output		
		
			// Check if TU which is nearer to the output is located higher in the stream	
			IF	mTU_Table[mTU_IdxOutput].DataSet.Sequence >  mTU_Table[mTU_IdxTemp].DataSet.Sequence OR 
				(mTU_Table[mTU_IdxOutput].DataSet.Sequence =  mTU_Table[mTU_IdxTemp].DataSet.Sequence AND
				mTU_Table[mTU_IdxOutput].DataSet.SubSequence >  mTU_Table[mTU_IdxTemp].DataSet.SubSequence)THEN				
				

				mSequenceErrorFound:= TRUE;
				EXIT;
				
			ELSE // TUs are in correct sequencing order
	
				// Set TU as new comparable
				mTU_IdxOutput := mTU_IdxTemp;
				TransportCtrlDataOutput:= TransportCtrlDataTemp;
			END_IF		
		END_IF
	END_IF
END_FOR


M_HasSquenceError:= mSequenceErrorFound;
END_METHOD

METHOD M_IsEmpty : BOOL // True = lane is empty, otherwise false
VAR
	mIdx				: DINT;
	mTransportCtrlData	: ST_TransportControlData;
END_VAR
M_IsEmpty:= TRUE;

// Loop through lane from outfeed to infeed
FOR mIdx:=1 TO PositionCount DO	
	
	mTransportCtrlData:= F_GetTransportControlData(Positions[mIdx].eFunctionNumber, Positions[mIdx].ZoneNumber);

	// Finish search when a TU was found		
	IF mTransportCtrlData.NumberOfPresentTUs > 0 THEN
		M_IsEmpty:= FALSE;
		EXIT;
	END_IF
	
END_FOR
END_METHOD

METHOD M_IsFull : BOOL // True = lane is full, otherwise false
VAR
	mIdx				: DINT;
	mTransportCtrlData	: ST_TransportControlData;
END_VAR
M_IsFull:= TRUE;

// Loop through lane from outfeed to infeed
FOR mIdx:=1 TO PositionCount DO	
	
	mTransportCtrlData:= F_GetTransportControlData(Positions[mIdx].eFunctionNumber, Positions[mIdx].ZoneNumber);

	// Finish search when a TU an empty zone was found	
	IF mTransportCtrlData.NumberOfPresentTUs = 0 THEN
		M_IsFull:= FALSE;
		EXIT;
	END_IF
	
END_FOR
END_METHOD

/// Check if TU may enter the lane, depening on  sequence information
METHOD M_RequestAccess : BOOL // True = Access granted, else false
VAR_INPUT
	mTU_Index			: DINT; // TU data index of requesting TU
END_VAR
VAR_IN_OUT 
	mTU_Table			: ARRAY[0..Conveyor.NUMBER_OF_TU_DATA] OF ST_TU_Data; // TU Table
END_VAR
VAR
	mIdx				: DINT;
	mTU_IndexLane		: DINT;
END_VAR
VAR_INST
	TransportCtrlData	: ST_TransportControlData;	
END_VAR
M_RequestAccess:=FALSE;	

IF M_IsEmpty() THEN

	// Grant access if TU has sequencing data or non sequencing TU's are allowed by configuration
	IF  mTU_Table[mTU_Index].DataSet.Sequence > 0 OR  NOT OnlySequencingTU THEN
		M_RequestAccess:=TRUE;	
	END_IF
	
ELSIF M_IsFull() THEN
	; //  Deny access

// Lane is partially full and requesting TU has no  sequencing data	
ELSIF  mTU_Table[mTU_Index].DataSet.Sequence = 0  THEN
		
	IF  NOT OnlySequencingTU THEN
		M_RequestAccess:= TRUE;
	END_IF

ELSE // Lane is partially full and requesting TU has data	
	
	// Search first TU after lane input with sequencing information
	FOR mIdx:=0 TO PositionCount-1 DO	

		TransportCtrlData:= F_GetTransportControlData(Positions[PositionCount-mIdx].eFunctionNumber, Positions[PositionCount-mIdx].ZoneNumber);
		mTU_IndexLane:= F_GetTU_DataIndex(Positions[PositionCount-mIdx].eFunctionNumber, Positions[PositionCount-mIdx].ZoneNumber);
	
		// Only consider TUs with whose Sequencing is not on hold
		IF TransportCtrlData.NumberOfPresentTUs > 0 AND 
			NOT mTU_Table[mTU_IndexLane].DataSet.HaltSequencing THEN
			
			 // Check if requesting TU is located higher in the stream (lower priority) than the found TU  
			IF  mTU_Table[mTU_Index].Destination[1].eFunctionNumber = mTU_Table[mTU_IndexLane].Destination[1].eFunctionNumber AND
				mTU_Table[mTU_Index].Destination[1].ZoneNumber = mTU_Table[mTU_IndexLane].Destination[1].ZoneNumber AND
				mTU_Table[mTU_Index].DataSet.DestinationSlot = mTU_Table[mTU_IndexLane].DataSet.DestinationSlot AND
				mTU_Table[mTU_Index].DataSet.Sequence >  mTU_Table[mTU_IndexLane].DataSet.Sequence OR 
				(mTU_Table[mTU_Index].DataSet.Sequence =  mTU_Table[mTU_IndexLane].DataSet.Sequence AND
				mTU_Table[mTU_Index].DataSet.SubSequence >  mTU_Table[mTU_IndexLane].DataSet.SubSequence)THEN	
								
				M_RequestAccess:= TRUE;				
			END_IF
			
			EXIT;	
			
		END_IF	
	END_FOR
END_IF
END_METHOD

// Only allow TU's to enter the lane which have sequencing data 
PROPERTY P_OnlySequencingTU : BOOL
GET
P_OnlySequencingTU:= OnlySequencingTU;
END_GET
SET
OnlySequencingTU:= P_OnlySequencingTU;
END_SET
END_PROPERTY

END_FUNCTION_BLOCK

// ---- 20_Product/30_Toolbox/17_WindowTracking/10_Core/FB_EncoderEx.TcPOU
/// Generates a synthetic encoder signal
// Remark: Can handle forward and reverese
FUNCTION_BLOCK FB_EncoderEx
(**************************************************************************************
 * 	Application		:	BoxControl Framework
 *	Revision		:	$Revision: 352787 $
 *	Revision date	:	$Date: 2015-07-23 08:18:11 +0200 (Do, 23 Jul 2015) $
 *	Last changed by	:	$Author: d7mangc $
 *	URL				:	$URL: http://almscdc.swisslog.com/repo/SWPD/Development/BoxControlFramework/20_Release/tags/R0.5.7/01_Software/BoxControlFramework/BoxControlFramework/JumpStart/11_Library/11Emulation/12_ElementFunctions/10_Functions/FB_TransportControlEmulation.TcPOU $
 *
 *	Purpose			:	Encoder 
 *
 * ------------------------------------------------------------------------------------
 *	Copyright Swisslog [IP AG], Switzerland. All rights reserved.
 * 
 * ------------------------------------------------------------------------------------
 *	
 * 	Revision History: 
 *
 * 	VERSION			DATE			INITIALS			DESCRIPTION
 *	0.1				01.01.2001		swl					Example
 *
 **************************************************************************************)
VAR_INPUT
	Run 			: BOOL; // Run command
	Speed 			: INT; // Speed [mm/s] + = Forward, - = Reverse
	RateIncPerMM 	: REAL := 1; // Encoder Resolution [Inc/mm]
	MaxEncoderValue	: UDINT; (* Max Encoder value
								Range = 0..MaxEncoderValue
							 *)
END_VAR
VAR_OUTPUT
	EncoderValue 	: UDINT; // Encoder value [Inc]
END_VAR
VAR
	Inc 			: DINT;
	IncLReal		: LREAL;
	Rest			: LREAL;
	EncoderValueDINT: DINT; // Encoder value [Inc]
	LastRest		: LREAL;
	LastSpeed   	: INT;
	t				: REAL;
	a				: REAL;
	StartCycl		: BOOL;
	fbGetCurTaskIdx : GETCURTASKINDEX;
	CycleTime       : UDINT;		
END_VAR

// Get current cycle time
fbGetCurTaskIdx();
CycleTime := _TaskInfo[fbGetCurTaskIdx.index].CycleTime;

// Calculate increment based on speed and resolution
IF Run THEN
	// t [s]
	t := (UDINT_TO_REAL(CycleTime) / 10000000.0);

	// Wait start cycle 
	IF StartCycl THEN
		// a = v - v0 / t [mm/s^2]
		a := (INT_TO_REAL(Speed - LastSpeed)) / t;	
	
		// Build result
		IncLReal := RateIncPerMM * (LastSpeed * t + 0.5 * a * EXPT(t,2));
		
		// Build rest *.x
		Rest := LMOD(IncLReal, 1) + LastRest;
		
		// Add trunc of rest
		IncLReal := IncLReal + LTRUNC(Rest);
		
		// Store last rest
		LastRest := LMOD(Rest, 1);
		
		// Incs s = v0 * t + 1/2 * a * t^2 [mm/s]
		// Remark: LTRUNG is used again to ensure the same rounding behavior
		Inc := LREAL_TO_DINT(LTRUNC(IncLReal));

		// Update last speed	
		LastSpeed := Speed;
	END_IF

	// Set start cycle done
	StartCycl := TRUE;
ELSE
	// Reset values
	StartCycl := FALSE;
	LastSpeed := 0;
	LastRest := 0;
	Inc := 0;
END_IF

// Update encoder value
EncoderValueDINT := EncoderValueDINT + Inc;

IF EncoderValueDINT > UDINT_TO_DINT(MaxEncoderValue) THEN
	EncoderValueDINT := EncoderValueDINT - (UDINT_TO_DINT(MaxEncoderValue) + 1); 
	
ELSIF EncoderValueDINT < 0 THEN
	EncoderValueDINT := UDINT_TO_DINT(MaxEncoderValue) + EncoderValueDint + 1;
END_IF

EncoderValue := DINT_TO_UDINT(EncoderValueDINT);

END_FUNCTION_BLOCK

// ---- 20_Product/30_Toolbox/17_WindowTracking/10_Core/FB_WindowRelocator.TcPOU
/// Handle relocation order in window tracking
{attribute 'no_explicit_call' := 'do not call this POU directly'} 
FUNCTION_BLOCK FB_WindowRelocator
(************************************************************************************** 
* 	Application 		: BoxControl Framework 
* 	Revision 			: $Revision: 408723 $ 
* 	Revision date 		: $Date: 2018-06-27 13:49:08 +0200 (Wed, 27 Jun 2018) $ 
* 	Last changed by 	: $Author: b7bolm $ 
* 	URL 				: $URL: http://almscdc.swisslog.com/repo/SWPD/Development/BoxControlFramework/21_Projects/BCF_2.0/trunk/BCF/BCF/JumpStart/20_Product/10_App/12_E_Functions/10_Lib/10_Conv/FB_FunctionList.TcPOU $ 
* ------------------------------------------------------------------------------------ 
* 	© Swisslog AG 
* 	Swisslog is not liable for any usage of this source code that is not agreed 
* 	on between Swisslog and the other party. The mandatory legal liability remains 
* 	unaffected. 
* ------------------------------------------------------------------------------------ 
* 	Revision History: 
* 
* 	VERSION 		DATE 			INITIALS 			DESCRIPTION 
* 	0.1 			31.08.2018 		b7bolm 				First implementation
* 
**************************************************************************************)
VAR
	Buffer  				: ARRAY[0..ENTRIES * UINT_TO_INT(SIZEOF(ST_WindowTrackingReloc))] OF BYTE; // Stack buffer
	fbReallocStack			: FB_MemStackBuffer; // Stack buffer LIFO
END_VAR
VAR CONSTANT
	ENTRIES 				: INT := 300; // Maximum index to store in buffer
	STACK_BUFFER_ERROR		: UINT := 1; // Error id for stack buffer
	MAX_NUMBER_OF_WINDOWS 	: UINT := WindowTracking.MAX_NUMBER_OF_WINDOWS;
	MAX_NUMBER_OF_ZONES		: UINT := MAX_NUMBER_OF_WINDOWS/2;
END_VAR

;

/// Clears all active orders
METHOD M_Reset : BOOL // Returns true if successful, otherwise false
M_Reset := FALSE;

fbReallocStack.A_Reset( 
	pBuffer 	:= ADR(Buffer), 
	cbBuffer 	:= SIZEOF(Buffer));
	
IF fbReallocStack.bOk THEN
	M_Reset := TRUE;
END_IF
END_METHOD

/// Returns last entred order
METHOD M_RetrieveLastEntry : BOOL // Returns true if an order could be successful retrieved.
VAR_INPUT
	mpData		: POINTER TO ST_WindowTrackingReloc; // Pointer to data variable
	mDataSize	: UINT; // Size of data variable
END_VAR
M_RetrieveLastEntry := FALSE;

IF fbReallocStack.nCount > 0 THEN
	// Retrieve and remove last
	fbReallocStack.A_Pop( 
		pBuffer 	:= ADR(buffer), 
		cbBuffer 	:= SIZEOF(buffer), 
		pRead 		:= mpData, 
		cbRead 		:= mDataSize);
		
	IF fbReallocStack.bOk THEN
		M_RetrieveLastEntry := TRUE;
	END_IF
END_IF
END_METHOD

/// Schedules a new reallocation of a window in WindowTracking
METHOD M_ScheduleRelocation : BOOL // Returns true, if reallocation was successful.
VAR_INPUT
	mZoneIndex				: UINT; // Zone index to reallocate
	mTargetWindow 			: UINT; // Target window to which the zone should be reallocated
	mMaxWindowIndex 		: UINT; // Maximum window index
	mrWindowTable			: REFERENCE TO ARRAY[1..MAX_NUMBER_OF_WINDOWS] OF ST_WindowTrackingWindow;
	mrZoneTable				: REFERENCE TO ARRAY[1..MAX_NUMBER_OF_ZONES] OF ST_WindowTrackingZone;
END_VAR
VAR_OUTPUT
	mBlockingZoneIndex 		: UINT;
	mBlockingEndWindowIndex : UINT;
	mErrorId				: UINT;
END_VAR
VAR_INST
	RelocOrder				: ST_WindowTrackingReloc; // Scheduled order
	RelocationPossible  	: BOOL; // Conditions allow reallocation 
	WindowLength 			: UINT; // Window length [windows] of a zone
END_VAR
VAR
	mIdx 					: UINT; // Iterator
	mWindowIndex 			: UINT; // Windes index iterator
	mTargetZoneIndex 		: UINT; // Target zone index
END_VAR
M_ScheduleRelocation := FALSE;
MEMSET(ADR(RelocOrder), 0, SIZEOF(RelocOrder));
RelocationPossible := TRUE;
mBlockingZoneIndex := 0;
mErrorId := 0;

IF mZoneIndex = 0 OR
   mTargetWindow = 0 OR
   NOT __ISVALIDREF(mrWindowTable) OR
   NOT __ISVALIDREF(mrZoneTable) THEN
   RETURN;
END_IF

IF mrZoneTable[mZoneIndex].ZoneEndWindowIndex > mrZoneTable[mZoneIndex].ZoneStartWindowIndex THEN
	WindowLength := mrZoneTable[mZoneIndex].ZoneEndWindowIndex - mrZoneTable[mZoneIndex].ZoneStartWindowIndex + 1;
ELSE
	WindowLength := mrZoneTable[mZoneIndex].ZoneEndWindowIndex + mMaxWindowIndex - mrZoneTable[mZoneIndex].ZoneStartWindowIndex + 1;
END_IF

mWindowIndex := mTargetWindow;

FOR mIdx := 1 TO WindowLength DO

	// Correct border overflow
	IF mWindowIndex > mMaxWindowIndex THEN
		mWindowIndex := mWindowIndex - mMaxWindowIndex;
	END_IF

	// Check if target window has already a reserved zone
	IF mrWindowTable[mWindowIndex].ZoneIndex <> 0 AND
        mrWindowTable[mWindowIndex].ZoneIndex <> mZoneIndex THEN
		// Store Zone index of target window
		mTargetZoneIndex := mrWindowTable[mWindowIndex].ZoneIndex;
	
		// Check if zone is allowed to be overwritten
		// - no physical TU is present
		// - shifting is not inhibited
		IF NOT mrZoneTable[mTargetZoneIndex].TU_Present AND
		   NOT mrZoneTable[mTargetZoneIndex].InhibitShifting THEN
		   // Window is possible to be overwritten, check others
		   ;
		ELSE
			RelocationPossible := FALSE;
			mBlockingZoneIndex := mTargetZoneIndex;
			mBlockingEndWindowIndex := mrZoneTable[mTargetZoneIndex].ZoneEndWindowIndex;
			EXIT;
		END_IF
	END_IF
	
	mWindowIndex := mWindowIndex + 1;
END_FOR

IF RelocationPossible THEN	
	RelocOrder.ZoneIndex := mZoneIndex;
	RelocOrder.TargetWindow := mTargetWindow;
	
	fbReallocStack.A_Push( 
		pBuffer 	:= ADR(Buffer),
		cbBuffer 	:= SIZEOF(Buffer),
		pWrite 		:= ADR(RelocOrder),
		cbWrite 	:= SIZEOF(RelocOrder));
		
	IF fbReallocStack.bOk THEN
		M_ScheduleRelocation := TRUE;
	ELSE
		mErrorId := STACK_BUFFER_ERROR;
		M_ScheduleRelocation := FALSE;	
	END_IF
END_IF
END_METHOD

/// Amount of available reallocation orders
{attribute 'monitoring' := 'call'}
PROPERTY P_Count : UDINT // Number of entries
GET
P_Count := fbReallocStack.nCount;
END_GET
END_PROPERTY

END_FUNCTION_BLOCK

// ---- 20_Product/30_Toolbox/17_WindowTracking/10_Core/FB_WindowTracking.TcPOU
/// Function block can manage multiple transport units of different lengths
FUNCTION_BLOCK FB_WindowTracking IMPLEMENTS I_WindowTracking
(************************************************************************************** 
* 	Application 		: BoxControl Framework 
* 	Revision 			: $Revision: 408723 $ 
* 	Revision date 		: $Date: 2018-06-27 13:49:08 +0200 (Wed, 27 Jun 2018) $ 
* 	Last changed by 	: $Author: b7bolm $ 
* 	URL 				: $URL: http://almscdc.swisslog.com/repo/SWPD/Development/BoxControlFramework/21_Projects/BCF_2.0/trunk/BCF/BCF/JumpStart/20_Product/10_App/12_E_Functions/10_Lib/10_Conv/FB_FunctionList.TcPOU $ 
* ------------------------------------------------------------------------------------ 
* 	© Swisslog AG 
* 	Swisslog is not liable for any usage of this source code that is not agreed 
* 	on between Swisslog and the other party. The mandatory legal liability remains 
* 	unaffected. 
* ------------------------------------------------------------------------------------ 
* 	Revision History: 
* 
* 	VERSION 		DATE 			INITIALS 			DESCRIPTION 
* 	0.1 			22.08.2018 		herzig 				First implementation
*	0.2				23.08.2018		mbo					Review
*	0.3				02.11.2018		mbo					Zone begin + end added
*														+ Listener extended
* 
**************************************************************************************)
VAR_INPUT
	EncoderValueInc			: UDINT; (* Current encoder value [inc] Ascending = forward *)
END_VAR
VAR_OUTPUT
	TrackingPosition		: UDINT; // Internal tracking position [mm]
	ZoneCount				: INT; // Number of allocated zones
	TU_Count				: INT; // Number of TUs on tracking
	WindowSize				: UINT := 100; // Size of windows [mm] Remark: Needs to be smaller than smallest transport unit
	TrackingLength			: UDINT; // Length of tracking segment [mm] (e.g. conveyor length)
	Initialized				: BOOL; // Module is initialized
END_VAR
VAR
	fbDebugMsg				: FB_DebugMsg; // Debug instance
	DebugMsg				: T_MAXSTRING; // Debug msg
	TrackingEncoderValue	: UDINT; // Internal tracking value
	RateIncPerMM			: LREAL; // Rate between increments and mm (How many increments represent one mm)
	MaxEncoderValueInc		: UDINT; // Max value of input "EncoderValue" [increments] Remark: Used to detect overflow
	TotalTrackingLength		: UDINT; // Complete tracking length
	TrackingAddition		: UDINT; // Tracking addition
	
	DeltaEncoderValue		: DINT; // Delta encoder value 
	DeleteZoneTrackingEnd	: BOOL := TRUE; // All zones get deleted on tracking end
	MaxWindowIndex			: UINT; // Max window index
	LastEncoderValueInc		: UDINT; // Encoder value of last cycle [increment]
	EndZoneIndex			: UINT; // Currently available zone index at conveyor end
	EndZoneStartPosition	: UDINT; // Start zone position of zone at conveyor end
	EndZoneEndPosition		: UDINT; // End zone position of zone at conveyor end
	EndWindowIndex			: UINT; // Window index at end of conveyor
	iEventListener			: I_WindowTrackingListener; // Tracking zone listener (0 = not used)
	LastDeletedEndZoneIndex	: UINT; // Last deleted index at tracking end, used for report
END_VAR

VAR CONSTANT
	MAX_MOVE_WINDOWS		: UINT := 200; // Maximum windows which can be stored temporarly
	TRANSFER_TABLE_SIZE		: UINT := 100; // Transfer table size
	MAX_NUMBER_OF_WINDOWS 	: UINT := WindowTracking.MAX_NUMBER_OF_WINDOWS;
	MAX_NUMBER_OF_ZONES		: UINT := MAX_NUMBER_OF_WINDOWS/2;
	DELAY_ZONE_LEFT_TRACKING	: UDINT := 5; //Small delay on deletion of the zones to ensure HandoverTracking deletes its TUs & zones first.
END_VAR

VAR PERSISTENT
	WindowTable				: ARRAY[1..MAX_NUMBER_OF_WINDOWS] OF ST_WindowTrackingWindow; // List of all windows
	ZoneTable				: ARRAY[1..MAX_NUMBER_OF_ZONES] OF ST_WindowTrackingZone; // List of all zones
	OngoingTransferList		: ARRAY[1..TRANSFER_TABLE_SIZE] OF ST_WindowTrackingTransfer; // TUs which are in transfer state to the tracking
	PTL_Zones				: ARRAY[1..MAX_NUMBER_OF_ZONES] OF UINT; // Zone to be monitored because of PositionToLive value
END_VAR

// Module needs to be initialized with required values
IF NOT Initialized THEN
	RETURN;
END_IF

// Generate encoder value
// ----------------------------------------------------
DeltaEncoderValue := UDINT_TO_DINT(EncoderValueInc) - UDINT_TO_DINT(LastEncoderValueInc);

IF ABS(DeltaEncoderValue) > UDINT_TO_DINT(MaxEncoderValueInc/2) THEN
	// Correction with + 1 is to include the 0 in MaxEncoderValue
	IF DeltaEncoderValue < 0 THEN
		DeltaEncoderValue := DeltaEncoderValue + UDINT_TO_DINT(MaxEncoderValueInc) + 1;
	ELSE
		DeltaEncoderValue := UDINT_TO_DINT(EncoderValueInc) - (UDINT_TO_DINT(LastEncoderValueInc) + UDINT_TO_DINT(MaxEncoderValueInc)) - 1;
	END_IF
END_IF

TrackingEncoderValue := DINT_TO_UDINT(UDINT_TO_DINT(TrackingEncoderValue) + DeltaEncoderValue);
 
LastEncoderValueInc := EncoderValueInc;

TrackingPosition := LREAL_TO_UDINT(UDINT_TO_LREAL(TrackingEncoderValue) / RateIncPerMM) MOD TotalTrackingLength;

// Manages ongoing transfers
// ----------------------------------------------------
M_ManageOngoingTransfers();

 // Manages position to live zones
// ----------------------------------------------------
M_MonitorZonesPTL();

// Delete all zones when they left the tracking length
// ----------------------------------------------------
IF DeleteZoneTrackingEnd THEN	
	IF EndZoneIndex > 0 THEN
		EndZoneStartPosition := M_GetZoneStartPosition(EndZoneIndex);
		EndZoneEndPosition := M_GetZoneEndPosition(EndZoneIndex);
		
		IF EndZoneStartPosition < TrackingLength + DELAY_ZONE_LEFT_TRACKING THEN
			EndZoneIndex := 0;
			
		ELSIF EndZoneEndPosition >= TrackingLength + DELAY_ZONE_LEFT_TRACKING THEN
			LastDeletedEndZoneIndex := EndZoneIndex;
			
			IF M_DeleteZone(EndZoneIndex) THEN
				// Zone deleted
				DebugMsg := CONCAT('Zone left tracking, zone deleted. ZoneIndex: ',UINT_TO_STRING(LastDeletedEndZoneIndex));;
				fbDebugMsg.M_SendInfoMsg(DebugMsg);
			ELSE
				DebugMsg := CONCAT('Zone left tracking, but could not be deleted. ZoneIndex: ',UINT_TO_STRING(LastDeletedEndZoneIndex));
				fbDebugMsg.M_SendErrorMsg(DebugMsg);
			END_IF
			
			EndZoneIndex := 0;
		END_IF
	ELSE
		EndZoneIndex := M_GetZoneIndex(TrackingLength);
		
		IF EndZoneIndex > 0 THEN
			DebugMsg := CONCAT('Zone index found at Tracking end. ZoneIndex: ',UINT_TO_STRING(EndZoneIndex));
			fbDebugMsg.M_SendInfoMsg(DebugMsg);
		END_IF
	END_IF
	
	// Delete all unassigned windows when they left the tracking length
	// ---------------------------------------------------- 
	EndWindowIndex := M_GetWindowIndex(TrackingLength);
	
	IF EndWindowIndex > 0 THEN
		IF WindowTable[EndWindowIndex].State <> E_WindowTrackingWindowState.IDLE THEN
			// Window has a valid ZoneIndex
			IF WindowTable[EndWindowIndex].ZoneIndex > 0 THEN
				// Check if its zone is still valid
				IF NOT ZoneTable[WindowTable[EndWindowIndex].ZoneIndex].Used THEN
					// Delete window
					M_ClearWindow(EndWindowIndex);
					
				// Check if window is inside zone start and end	
				ELSE
					IF ZoneTable[WindowTable[EndWindowIndex].ZoneIndex].ZoneEndWindowIndex >= ZoneTable[WindowTable[EndWindowIndex].ZoneIndex].ZoneStartWindowIndex THEN
						IF EndWindowIndex < ZoneTable[WindowTable[EndWindowIndex].ZoneIndex].ZoneStartWindowIndex OR
				   		   EndWindowIndex > ZoneTable[WindowTable[EndWindowIndex].ZoneIndex].ZoneEndWindowIndex THEN
						   	// Delete window
							M_ClearWindow(EndWindowIndex);
						END_IF		
					ELSE
						IF EndWindowIndex < ZoneTable[WindowTable[EndWindowIndex].ZoneIndex].ZoneStartWindowIndex AND
				   		   EndWindowIndex > ZoneTable[WindowTable[EndWindowIndex].ZoneIndex].ZoneEndWindowIndex THEN
						   	// Delete window
							M_ClearWindow(EndWindowIndex);
						END_IF
					END_IF
				END_IF
			ELSE
				// Delete window
				M_ClearWindow(EndWindowIndex);
			END_IF
		END_IF
	END_IF
END_IF

/// Adds a TU to the beginning of the zone
METHOD M_AddTU : BOOL // Returns true successfully, otherwise false (Zone not found, Zone to small or already occupied)
VAR_INPUT
	mZoneIndex				: UINT;	// Zone index 
	mTU_Index				: DINT; // Index of TU to add
	mLength					: UINT; // Length of TU to be added [mm] Remark: Needs to be > than WindowSize
	mTU_Offset				: UINT; // Relative TU offset position in zone [mm]
END_VAR
VAR
	mIdx					: UINT; // Loop iterator
	mWindowIndex			: UINT; // Window index interator
	mNumberLengthWindows	: UINT; // Number of windows to allocate
	mRelWindowPositionFE	: UDINT; // Relative position in first window
	mRelWindowPositionRE	: UDINT; // Relative position in last window
	mFullLength				: UINT; // Complete length which is required from window begin
	mTU_OffsetWindows		: UINT; // TU offset in number of windows
END_VAR
M_AddTU := FALSE;

// Validate inputs
IF mZoneIndex = 0 OR 
   mZoneIndex > MAX_NUMBER_OF_ZONES OR
   mLength = 0 OR 
   mLength > TrackingLength OR
   mLength <= WindowSize OR
   WindowSize = 0 THEN
	RETURN;
END_IF

// When zone is not used, already occupied or too small, abort
IF NOT ZoneTable[mZoneIndex].Used OR
   ZoneTable[mZoneIndex].TU_Present OR
   mLength > ZoneTable[mZoneIndex].ZoneLength THEN
   RETURN;
END_IF

// Calculate relative position in first zone window
IF ZoneTable[mZoneIndex].ZoneStartPosition + mTU_Offset <= TotalTrackingLength THEN
	mRelWindowPositionFE := (ZoneTable[mZoneIndex].ZoneStartPosition + mTU_Offset) MOD WindowSize;
ELSE
	mRelWindowPositionFE := (ZoneTable[mZoneIndex].ZoneStartPosition + mTU_Offset - TotalTrackingLength) MOD WindowSize;
END_IF

// The relative position in the first window is added to the length, 
// in order to get the amount of windows which are allocated for that TU finally
mFullLength := mLength + UDINT_TO_UINT(mRelWindowPositionFE);

// Convert length into number of windows
mNumberLengthWindows := mFullLength / WindowSize;
// If not the full length could be mapped in windows
// add an additional window
IF (mFullLength MOD WindowSize) > 0 THEN
	mNumberLengthWindows := mNumberLengthWindows + 1;
END_IF

// Convert TU_Offset into number of windows
mTU_OffsetWindows := mTU_Offset / WindowSize;

mWindowIndex := ZoneTable[mZoneIndex].ZoneStartWindowIndex;

ZoneTable[mZoneIndex].TU_Present := TRUE;
ZoneTable[mZoneIndex].TU_Index := mTU_Index;
TU_Count := TU_Count + 1;

// First, the whole TU is added to the beginning of the window of the front edge window
FOR mIdx := 1 TO mNumberLengthWindows + mTU_OffsetWindows DO
	// Set start edge of TU to zone begin
	IF mIdx = mTU_OffsetWindows + 1 THEN
		WindowTable[mWindowIndex].State := E_WindowTrackingWindowState.FRONT_EDGE;
		WindowTable[mWindowIndex].TU_FrontEdgePosition := ZoneTable[mZoneIndex].ZoneStartPosition + mTU_Offset;
		
		ZoneTable[mZoneIndex].TU_StartWindowIndex := mWindowIndex;

	ELSIF mIdx = mNumberLengthWindows + mTU_OffsetWindows THEN
		// Length -1 is correction of window 
		// Example: Window1 has the following range 0..WindowSize-1
		mRelWindowPositionRE := (mFullLength - 1) MOD WindowSize;
		WindowTable[mWindowIndex].State := E_WindowTrackingWindowState.REAR_EDGE;
		
		ZoneTable[mZoneIndex].TU_EndWindowIndex := mWindowIndex;
		
		WindowTable[mWindowIndex].TU_RearEdgePosition := mRelWindowPositionRE + (mWindowIndex - 1) * WindowSize;
		
	ELSIF mIdx > mTU_OffsetWindows + 1 THEN
		WindowTable[mWindowIndex].State := E_WindowTrackingWindowState.OCCUPIED;
	END_IF
	
	mWindowIndex := mWindowIndex + 1;

	// Correct window border overflow
	IF mWindowIndex > MaxWindowIndex THEN
		mWindowIndex := mWindowIndex - MaxWindowIndex;
	END_IF
END_FOR

// Inform listener
IF iEventListener <> 0 THEN
	iEventListener.M_TrackingTU_AddedEvent(mZoneIndex, ZoneTable[mZoneIndex]);
END_IF

// Notify listener about change of TU state
IF ZoneTable[mZoneIndex].iActionListener <> 0 THEN
	ZoneTable[mZoneIndex].iActionListener.M_ActionZoneChangedEvent(mZoneIndex, ZoneTable[mZoneIndex]);
END_IF

M_AddTU := TRUE;
END_METHOD

/// Adds a TU to the tracking by creating a Zone and setting the front edge.
/// The add process is completed by triggering M_AddTU_RearEdge
METHOD M_AddTU_FE : UINT // Returns ZoneIndex > 0 if successfully, otherwise 0
VAR_INPUT
	mTU_Index				: DINT; // Index of TU to add
	mAbsolutePosition		: UDINT; // Position where a TU should be added
	miActionListener		: I_TrackingActionListener; // Action listener of the created zone
END_VAR
VAR_INST
	ZoneIndex				: UINT; // New zone index
	WindowIndex				: UINT; // Actual window index
END_VAR
VAR
	mIdx					: UINT; // Loop iterator
	mFreeOK					: BOOL; // Shift operation successful
	mShortenOK				: BOOL; // Shorten operation successful
	mTrackingPosition		: UDINT; // Position of TU on tracking
	mZoneLength				: UDINT; // Allocated zone length
END_VAR
// Initialize
ZoneIndex := 0;
M_AddTU_FE := 0;
mShortenOK := FALSE;

// Get window of absolute position
WindowIndex := M_GetWindowIndex(mAbsolutePosition);

IF WindowIndex > 0 AND WindowIndex <= WindowTracking.MAX_NUMBER_OF_WINDOWS THEN	
	// Is on intended window index already part of a zone, try to shift
	IF WindowTable[WindowIndex].ZoneIndex > 0 THEN
		// Make space
		mFreeOK := M_MakeSpaceByWindows(mAbsolutePosition, 1, TRUE);
	END_IF
	
	// Get a free zone index
	ZoneIndex := M_InsertNewZoneIndex();
	
	IF ZoneIndex > 0 THEN
		// Clear window
		MEMSET(ADR(WindowTable[WindowIndex]), 0, SIZEOF(WindowTable[WindowIndex]));
		
		// Get position on tracking
		mTrackingPosition := M_GetTrackingPosition(mAbsolutePosition);
	
		// Fill out window of front edge
		WindowTable[WindowIndex].State := E_WindowTrackingWindowState.FRONT_EDGE;
		WindowTable[WindowIndex].TU_FrontEdgePosition := mTrackingPosition;
		WindowTable[WindowIndex].ZoneIndex := ZoneIndex;
		
		TU_Count := TU_Count + 1;
		
		// TU gets inserted in a "transfer list" to keep assigning
		// upcoming windows until transport is completed.
		FOR mIdx := 1 TO TRANSFER_TABLE_SIZE DO
			// Search an empty slot
			IF NOT OngoingTransferList[mIdx].Active THEN
				OngoingTransferList[mIdx].Active := TRUE;
				OngoingTransferList[mIdx].AbsoluteInsertPosition := mAbsolutePosition;
				OngoingTransferList[mIdx].ZoneIndex := ZoneIndex;
				OngoingTransferList[mIdx].LastWindowIndex := WindowIndex;
				EXIT;
			END_IF
		END_FOR
		
		// Get used zone length from start point to end of first window
		mZoneLength := WindowSize - (mTrackingPosition MOD WindowSize);
		
		// Update zone information
		ZoneTable[ZoneIndex].TU_Present := TRUE;
		ZoneTable[ZoneIndex].TU_Index := mTU_Index;
		ZoneTable[ZoneIndex].iActionListener := miActionListener;
		ZoneTable[ZoneIndex].ZoneStartWindowIndex := WindowIndex;
		ZoneTable[ZoneIndex].TU_StartWindowIndex := WindowIndex;
		ZoneTable[ZoneIndex].ZoneStartPosition := mTrackingPosition;
		ZoneTable[ZoneIndex].ZoneEndWindowIndex := WindowIndex;
		ZoneTable[ZoneIndex].TU_EndWindowIndex := WindowIndex;
		ZoneTable[ZoneIndex].ZoneEndPosition := WindowIndex * WindowSize - 1;
		
		ZoneTable[ZoneIndex].ZoneLength := UDINT_TO_UINT(mZoneLength);
		
		// Inform listener
		IF iEventListener <> 0 THEN
			iEventListener.M_TrackingZoneAddedEvent(ZoneIndex,ZoneTable[ZoneIndex]);
		END_IF
		
		M_AddTU_FE := ZoneIndex;
	ELSE
		// Error no free zones anymore
		fbDebugMsg.M_SendErrorMsg('M_AddTU_FE - Could not allocated new zone');
		M_AddTU_FE := 0;
	END_IF
END_IF
END_METHOD

/// Completes an AddTU process which was initiated by M_AddTU_FrontEdge
/// Remark: Founds between FE and RE would be deleted automatically
METHOD M_AddTU_RE : UINT // Returns ZoneIndex > 0 if successfully, otherwise 0
VAR_INPUT
	mAbsolutePosition		: UDINT; // Position where a TU should be added
	mZoneIndex				: UINT;	// Zone index to be completed
END_VAR
VAR_INST
	WindowIndex				: UINT; // Window index of absolute position
END_VAR
VAR
	mIdx					: UINT; // Loop iterator
	mFreeOk					: BOOL; // Shift operation successful
	mTrackingPosition		: UDINT; // Position of TU on tracking
	mZoneFound				: BOOL; // Zone is part of transfer list
	mWindowLength			: UINT; // Windows length
	mWindowIndex			: UINT; // Window index interator
	mDeletedOnTransferList	: BOOL; // Zone was found and deleted on transfer list
END_VAR
M_AddTU_RE := 0;

// Validate inputs
IF mZoneIndex = 0 OR 
   mZoneIndex > MAX_NUMBER_OF_ZONES THEN
	RETURN;
END_IF

// Ensure that Zone index is available
FOR mIdx := 1 TO TRANSFER_TABLE_SIZE DO
	IF OngoingTransferList[mIdx].Active THEN	
		IF OngoingTransferList[mIdx].ZoneIndex = mZoneIndex THEN 
			mZoneFound := TRUE;
		END_IF
	ELSE
		// No entries available
		EXIT;
	END_IF
END_FOR

// When zone is part of transfer list, update rear edge
IF mZoneFound THEN
	// Calculate window index of absolute position
	WindowIndex := M_GetWindowIndex(mAbsolutePosition);
	
	IF WindowIndex > 0 AND WindowIndex <= WindowTracking.MAX_NUMBER_OF_WINDOWS THEN
		// Is on intended window index already part of a zone, try to shift
		IF WindowTable[WindowIndex].ZoneIndex > 0 AND 
		   WindowTable[WindowIndex].ZoneIndex <> mZoneIndex THEN
			// Shift reserved zones
			mFreeOK := M_MakeSpaceByWindows(mAbsolutePosition, 1, TRUE);
		END_IF
		
		// Ensure rear edge window is no front edge window, otherwise invalid -> Abort and delete
		IF WindowTable[WindowIndex].State = E_WindowTrackingWindowState.FRONT_EDGE THEN
			IF M_DeleteZone(mZoneIndex) THEN
				DebugMsg := CONCAT('M_AddTU_RE - Front edge window found -> Invalid. Zone deleted. Zone index: ',UINT_TO_STRING(mZoneIndex));
				fbDebugMsg.M_SendInfoMsg(DebugMsg);
			ELSE
				DebugMsg := CONCAT('M_AddTU_RE - Front edge window found -> Invalid. Deleting of zone failed . Zone index: ',UINT_TO_STRING(mZoneIndex));
				fbDebugMsg.M_SendErrorMsg(DebugMsg);
			END_IF	
			M_AddTU_RE := 0;
			RETURN;
		END_IF
		
		// Clear window
		MEMSET(ADR(WindowTable[WindowIndex]), 0, SIZEOF(WindowTable[WindowIndex]));
	
		// Get position on tracking
		mTrackingPosition := M_GetTrackingPosition(mAbsolutePosition);
		
		// Update window
		WindowTable[WindowIndex].ZoneIndex := mZoneIndex;
		WindowTable[WindowIndex].State := E_WindowTrackingWindowState.REAR_EDGE;
		WindowTable[WindowIndex].TU_RearEdgePosition := mTrackingPosition;
		
		// Clean entry in transfer list and close gaps in list
		mDeletedOnTransferList := M_RemoveZoneFromTransferList(mZoneIndex);
		
		// Update zone data
		ZoneTable[mZoneIndex].ZoneEndWindowIndex := WindowIndex;
		ZoneTable[mZoneIndex].TU_EndWindowIndex := WindowIndex;
		ZoneTable[mZoneIndex].ZoneEndPosition := mTrackingPosition;
		
		IF ZoneTable[mZoneIndex].ZoneEndPosition >= ZoneTable[mZoneIndex].ZoneStartPosition THEN
			ZoneTable[mZoneIndex].ZoneLength := UDINT_TO_UINT(ZoneTable[mZoneIndex].ZoneEndPosition - ZoneTable[mZoneIndex].ZoneStartPosition);
		ELSE
			ZoneTable[mZoneIndex].ZoneLength := UDINT_TO_UINT(ZoneTable[mZoneIndex].ZoneEndPosition + TotalTrackingLength - ZoneTable[mZoneIndex].ZoneStartPosition);
		END_IF
		
		// Check if all windows between Start and Endwindow are occupied and assigned to this zone index
		mWindowIndex := ZoneTable[mZoneIndex].TU_StartWindowIndex;
		
		IF ZoneTable[mZoneIndex].TU_EndWindowIndex >= ZoneTable[mZoneIndex].TU_StartWindowIndex THEN
			mWindowLength :=ZoneTable[mZoneIndex].TU_EndWindowIndex - ZoneTable[mZoneIndex].TU_StartWindowIndex + 1;
		ELSE
			mWindowLength :=ZoneTable[mZoneIndex].TU_EndWindowIndex + MaxWindowIndex  - ZoneTable[mZoneIndex].TU_StartWindowIndex + 1;
		END_IF
		
		FOR mIdx := 1 TO mWindowLength DO
			IF WindowTable[mWindowIndex].ZoneIndex = 0 THEN
				// Update window
				WindowTable[mWindowIndex].State := E_WindowTrackingWindowState.OCCUPIED;
				WindowTable[mWindowIndex].ZoneIndex := mZoneIndex;
							
			ELSIF WindowTable[mWindowIndex].ZoneIndex <> mZoneIndex THEN 
				// Something went wrong, other zone found between start and end window
				DebugMsg := CONCAT('M_AddTU_RE - Other zone found between start and end window of zone:',UINT_TO_STRING(mZoneINdex));
				fbDebugMsg.M_SendErrorMsg(DebugMsg);
			END_IF
			
			mWindowIndex := mWindowIndex + 1;
			
			// Correct window border overflow
			IF mWindowIndex > MaxWindowIndex THEN
				mWindowIndex := mWindowIndex - MaxWindowIndex;
			END_IF
		END_FOR
	
		// Inform listener
		IF iEventListener <> 0 THEN
			iEventListener.M_TrackingTU_AddedEvent(mZoneIndex,ZoneTable[mZoneIndex]);
		END_IF
		
		M_AddTU_RE := mZoneIndex;
	END_IF
// Zone is not part of transfer  list
ELSE
	fbDebugMsg.M_SendErrorMsg('M_AddTU_RE - Zone is not in transfer (not part of ongoing transfers)');
END_IF
END_METHOD

/// Adds a zone to the PTL list, so the zone PTL gets monitored
METHOD PROTECTED M_AddZoneToPTL : BOOL // Returns true if successfully added, otherwise false
VAR_INPUT
	mZoneIndex			: UINT; // Zone index to add
END_VAR
VAR
	mIdx				: UINT; // Iterator
END_VAR
M_AddZoneToPTL := FALSE;

// Validate inputs
IF mZoneIndex = 0 OR 
   mZoneIndex > MAX_NUMBER_OF_ZONES THEN
	RETURN;
END_IF

// When zone is not in used or already occupied, abort
IF NOT ZoneTable[mZoneIndex].Used OR
   ZoneTable[mZoneIndex].TU_Present THEN
   RETURN;
END_IF

// TU gets inserted in a list to be monitored PTL
FOR mIdx := 1 TO MAX_NUMBER_OF_ZONES DO
	// Search an empty slot or same
	IF PTL_Zones[mIdx] = 0 OR 
       PTL_Zones[mIdx] = mZoneIndex THEN
		PTL_Zones[mIdx] := mZoneIndex;
		M_AddZoneToPTL := TRUE;
		EXIT;
	END_IF
END_FOR
END_METHOD

/// Adjust front edge position inside a front edge window and aligns rear edge accordingly. 
/// Remark: TU Length stays the same, but its possible that number of used windows is changing.
/// Remark: Found zones at target get shifted or deleted according configuration
METHOD PROTECTED M_AdjustFE : BOOL // Returns true if successfully adjusted, otherwise false (e.g. no front edge window)
VAR_INPUT
	mWindowIndexFE			: UINT; // Window index of front edge
	mNewTrackingPosition	: UDINT; // Tracking position to which the edge should be moved to [mm]
	mDeleteTargetZones  	: BOOL; // Zones at target destination gets deleted, otherwise shifted
END_VAR
VAR
	mZoneDeleted 			: BOOL; // Zone at target was deleted successfully
	mZoneOk 				: BOOL; // Zone at target was shifted successfully
END_VAR
VAR_INST
	UpdateZoneEndWindowIndex: BOOL; // UpdateZoneEndWindowIndex
	ZoneIndex 				: UINT; // Found zone index
	ZoneWindowLength 		: UINT; // Length of zone in windows
	MovePossible 			: BOOL; // Move valid
	MaxWindowPosition 		: UDINT; // Input check for required poition MAX
	MinWindowPosition 		: UDINT; // Input check for required poition MIN
	OldRelWindowPositionFE 	: UDINT; // Old relative window position front edge
	OldRelWindowPositionRE 	: UDINT; // Old relative window position rear edge
	WindowIndexRE			: UINT; // Window index rear edge
	NewWindowIndexRE 		: UINT; // New window index rear edge
	NewRelWindowPositionFE 	: UDINT; // New relative window position front edge
	NewRelWindowPositionRE 	: DINT; // New relative window position rear edge
	NewAbsWindowPositionRE 	: UDINT; // New absolute window position rear edge
	DeltaWindowPositionFE 	: DINT; // Delte distance of edge movement
END_VAR
// Initialize
M_AdjustFE := FALSE;
UpdateZoneEndWindowIndex := FALSE;
ZoneIndex := 0;
ZoneWindowLength := 0;
WindowIndexRE := 0;

// Validate inputs
IF mWindowIndexFE = 0 OR
   mWindowIndexFE > MaxWindowIndex  THEN
   RETURN;
END_IF

// Get max and min tracking position of front edge window
MaxWindowPosition := (mWindowIndexFE) * WindowSize;
MinWindowPosition := (mWindowIndexFE-1) * WindowSize;

// Ensure that new tracking position is in range of window
IF mNewTrackingPosition < MinWindowPosition OR 
   mNewTrackingPosition >= MaxWindowPosition THEN
   RETURN;
END_IF

// Try to get the corresponding zone and ensure its valid
IF WindowTable[mWindowIndexFE].State <> E_WindowTrackingWindowState.FRONT_EDGE OR 
   WindowTable[mWindowIndexFE].ZoneIndex = 0 THEN
	RETURN;
END_IF

ZoneIndex := WindowTable[mWindowIndexFE].ZoneIndex;

// Calculate length of zone in windows
IF ZoneTable[ZoneIndex].ZoneEndWindowIndex > ZoneTable[ZoneIndex].ZoneStartWindowIndex THEN
	ZoneWindowLength := ZoneTable[ZoneIndex].ZoneEndWindowIndex - ZoneTable[ZoneIndex].ZoneStartWindowIndex + 1;
ELSE
	ZoneWindowLength := ZoneTable[ZoneIndex].ZoneEndWindowIndex + MaxWindowIndex  - ZoneTable[ZoneIndex].ZoneStartWindowIndex + 1;
END_IF

// Update front edge position
OldRelWindowPositionFE := WindowTable[mWindowIndexFE].TU_FrontEdgePosition MOD WindowSize;
WindowTable[mWindowIndexFE].TU_FrontEdgePosition := mNewTrackingPosition;

// When Zone begin is same as Frontedge window
IF ZoneTable[ZoneIndex].ZoneStartWindowIndex = mWindowIndexFE THEN
	// Check if adjustment of TU front edge would enlarge zone
	IF ZoneTable[ZoneIndex].ZoneStartPosition > mNewTrackingPosition THEN
		// Adjust zone begin
		ZoneTable[ZoneIndex].ZoneStartPosition := mNewTrackingPosition;
	END_IF
END_IF

//Get rear edge window index
WindowIndexRE := ZoneTable[ZoneIndex].TU_EndWindowIndex;

// When no rear edge could be found
IF WindowIndexRE = 0 THEN
	// Failed
	M_AdjustFE := FALSE;
	RETURN;
END_IF

// Get difference between old and new position in window
NewRelWindowPositionFE := mNewTrackingPosition MOD WindowSize;

DeltaWindowPositionFE := UDINT_TO_DINT(NewRelWindowPositionFE) 
						 - UDINT_TO_DINT(OldRelWindowPositionFE);

OldRelWindowPositionRE := WindowTable[WindowIndexRE].TU_RearEdgePosition MOD WindowSize;

// Calculate relative TU position in new window
NewRelWindowPositionRE := UDINT_TO_DINT(OldRelWindowPositionRE) + DeltaWindowPositionFE;

MovePossible := TRUE;

// When new position in window is more than one window -> additional window required
IF NewRelWindowPositionRE >= WindowSize THEN
	NewWindowIndexRE := WindowIndexRE + 1;
	
	IF NewWindowIndexRE > MaxWindowIndex THEN
		NewWindowIndexRE := NewWindowIndexRE - MaxWindowIndex;
	END_IF
	
	// Check if this window consists already of a zone
	IF WindowTable[NewWindowIndexRE].ZoneIndex > 0 THEN
		IF WindowTable[NewWindowIndexRE].ZoneIndex <> ZoneIndex THEN
		   // A new window is required which was not part of this zone before (No window with reservation state)
		   UpdateZoneEndWindowIndex := TRUE;
		   
			// If another zone is found, try to shift / delete it
		   IF mDeleteTargetZones THEN
				mZoneDeleted := M_DeleteZone(WindowTable[NewWindowIndexRE].ZoneIndex);
				
				IF NOT mZoneDeleted THEN
					// Error, zone could not be deleted -> abort
					MovePossible := FALSE;
				END_IF
			ELSE
				// Otherwise make space
				mZoneOk :=	M_MakeSpace(
								mStartWindowIndex 	:= NewWindowIndexRE, 
								mWindowsToFree 		:= 1,
								mAllowZoneDelete 	:= TRUE);
												
				IF NOT mZoneOk THEN
					// Error, zone could not be shifted -> abort
					MovePossible := FALSE;
				END_IF
			END_IF
		END_IF
	ELSE
		// A new window is required which was not part of this zone before (No window with reservation state)
		UpdateZoneEndWindowIndex := TRUE;
	END_IF
	
	// If zone of new needed window can not be moved, edge can not be adjusted
	IF NOT MovePossible THEN
		// Move not possible, adjustment failed
		M_AdjustFE := FALSE;
		RETURN;
	END_IF
	
	// If a new window was required to be allocated, update end window index
	IF UpdateZoneEndWindowIndex THEN
		ZoneTable[ZoneIndex].ZoneEndWindowIndex := NewWindowIndexRE;
	END_IF 
	
	// Copy window
	WindowTable[NewWindowIndexRE] := WindowTable[WindowIndexRE];
	
	ZoneTable[ZoneIndex].TU_EndWindowIndex := NewWindowIndexRE;
	
	// Clear exiting rear edge window
	M_ClearWindow(WindowIndexRE);
	
	// Assign window between occupied and takeover same flags
	WindowTable[WindowIndexRE].State := E_WindowTrackingWindowState.OCCUPIED;
	WindowTable[WindowIndexRE].ZoneIndex := ZoneIndex;
	WindowTable[WindowIndexRE].Flush := ZoneTable[ZoneIndex].Flush;

// When new position in window is less than 0 -> one window can be removed
ELSIF NewRelWindowPositionRE < 0 THEN
	NewWindowIndexRE := WindowIndexRE - 1;
	
	IF NewWindowIndexRE <= 0 THEN
		NewWindowIndexRE := NewWindowIndexRE + MaxWindowIndex;
	END_IF
	
	// Copy window
	WindowTable[NewWindowIndexRE] := WindowTable[WindowIndexRE];
	
	ZoneTable[ZoneIndex].TU_EndWindowIndex := NewWindowIndexRE;
	
	// If old window was end of zone, clear window, otherwise mark as reserved 
	// beacuse it is still part of the zone but not of the TU anymore
	IF WindowIndexRE = ZoneTable[ZoneIndex].ZoneEndWindowIndex THEN
		// Clear window
		M_ClearWindow(WindowIndexRE);
		
		ZoneTable[ZoneIndex].ZoneEndWindowIndex := NewWindowIndexRE;
	ELSE
		WindowTable[WindowIndexRE].TU_RearEdgePosition := 0;
		WindowTable[WindowIndexRE].State := E_WindowTrackingWindowState.RESERVED;
	END_IF
		
// Window index stays the same
ELSE
	NewWindowIndexRE := WindowIndexRE;
END_IF 

// Correct rear edge and update window and zone
NewAbsWindowPositionRE := DINT_TO_UDINT(NewRelWindowPositionRE) MOD WindowSize + 
					  	  (NewWindowIndexRE -1)*WindowSize;

WindowTable[NewWindowIndexRE].TU_RearEdgePosition := NewAbsWindowPositionRE;

// If rear edge window is last in zone, check position inside window
IF NewWindowIndexRE = ZoneTable[ZoneIndex].ZoneEndWindowIndex THEN
	// Check if adjustment of TU rear edge would enlarge zone and adapt
	// REMARK: Reduce the length of zone is not allowed, because this could have influence to 
    // minimum gaps between zones
	IF ZoneTable[ZoneIndex].ZoneEndPosition < WindowTable[NewWindowIndexRE].TU_RearEdgePosition THEN
		// Adjust zone end
		ZoneTable[ZoneIndex].ZoneEndPosition := WindowTable[NewWindowIndexRE].TU_RearEdgePosition;
	END_IF
END_IF

// Calculate new length
IF ZoneTable[ZoneIndex].ZoneEndPosition >= ZoneTable[ZoneIndex].ZoneStartPosition THEN
	ZoneTable[ZoneIndex].ZoneLength := UDINT_TO_UINT(ZoneTable[ZoneIndex].ZoneEndPosition 
															   - ZoneTable[ZoneIndex].ZoneStartPosition);
ELSE
	ZoneTable[ZoneIndex].ZoneLength := UDINT_TO_UINT(ZoneTable[ZoneIndex].ZoneEndPosition 
															  + TotalTrackingLength 
															  - ZoneTable[ZoneIndex].ZoneStartPosition);
END_IF

M_AdjustFE := TRUE;
END_METHOD

/// Adjust rear edge position inside a rear edge window and aligns front edge accordingly. 
/// Remark: TU Length stays the same, but its possible that number of used windows is changing.
/// Remark: Found zones at target get shifted or deleted according configuration
METHOD PROTECTED M_AdjustRE : BOOL // Returns true if successfully adjusted, otherwise false (e.g. no rear edge window)
VAR_INPUT
	mWindowIndexRE				: UINT; // Window index of rear edge
	mNewTrackingPosition		: UDINT; // Tracking position to which the edge should be moved to [mm]
	mDeleteTargetZones  		: BOOL; // Zones at target destination gets deleted, otherwise shifted
END_VAR
VAR_INST
	ZoneIndex 					: UINT; // Found zone index
	ZoneWindowLength 			: UINT; // Length of zone in windows
	UpdateZoneStartWindowIndex 	: BOOL; // Adjustment required an additional window
	MovePossible 				: BOOL; // Move valid
	MaxWindowPosition 			: UDINT; // Input check for required poition MAX
	MinWindowPosition	    	: UDINT; // Input check for required poition MIN
	OldRelWindowPositionFE 		: UDINT; // Old relative window position front edge
	OldRelWindowPositionRE 		: UDINT; // Old relative window position rear edge
	WindowIndexFE				: UINT; // Window index front edge
	NewWindowIndexFE 			: UINT; // New window index rear edge
	NewRelWindowPositionRE 		: UDINT; // New relative window position rear edge
	NewRelWindowPositionFE 		: DINT; // New relative window position front edge
	NewAbsWindowPositionFE 		: UDINT; // New absolute window position front edge
	DeltaWindowPositionRE 		: DINT; // Delte distance of edge movement
END_VAR
// Initialize
M_AdjustRE := FALSE;
UpdateZoneStartWindowIndex := FALSE;
ZoneIndex := 0;
ZoneWindowLength := 0;
WindowIndexFE := 0;

// Validate inputs
IF mWindowIndexRE = 0 OR
   mWindowIndexRE > MaxWindowIndex  THEN
   RETURN;
END_IF

// Get max and min tracking position of front edge window
MaxWindowPosition := (mWindowIndexRE) * WindowSize;
MinWindowPosition := (mWindowIndexRE-1) * WindowSize;

// Ensure that new tracking position is in range of window
IF mNewTrackingPosition < MinWindowPosition OR 
   mNewTrackingPosition >= MaxWindowPosition THEN
   RETURN;
END_IF

// Try to get the corresponding zone and ensure its valid
IF WindowTable[mWindowIndexRE].State <> E_WindowTrackingWindowState.REAR_EDGE OR 
   WindowTable[mWindowIndexRE].ZoneIndex = 0 THEN
	RETURN;
END_IF

ZoneIndex := WindowTable[mWindowIndexRE].ZoneIndex;

// Calculate length of zone in windows
IF ZoneTable[ZoneIndex].ZoneEndWindowIndex > ZoneTable[ZoneIndex].ZoneStartWindowIndex THEN
	ZoneWindowLength := ZoneTable[ZoneIndex].ZoneEndWindowIndex - ZoneTable[ZoneIndex].ZoneStartWindowIndex + 1;
ELSE
	ZoneWindowLength := ZoneTable[ZoneIndex].ZoneEndWindowIndex + MaxWindowIndex  - ZoneTable[ZoneIndex].ZoneStartWindowIndex + 1;
END_IF

// Update rear edge position
OldRelWindowPositionRE := WindowTable[mWindowIndexRE].TU_RearEdgePosition MOD WindowSize;
WindowTable[mWindowIndexRE].TU_RearEdgePosition := mNewTrackingPosition;

// When Zone end is same as Rearedge window
IF ZoneTable[ZoneIndex].ZoneEndWindowIndex = mWindowIndexRE THEN
	// Check if adjustment of TU rear edge would enlarge zone
	IF ZoneTable[ZoneIndex].ZoneEndPosition < mNewTrackingPosition THEN
		// Adjust zone end
		ZoneTable[ZoneIndex].ZoneEndPosition := mNewTrackingPosition;
	END_IF
END_IF

// Get window index of front edge
WindowIndexFE := ZoneTable[ZoneIndex].TU_StartWindowIndex;

// When no front edge could be found
IF WindowIndexFE = 0 THEN
	// Failed
	M_AdjustRE := FALSE;
	RETURN;
END_IF

// Get difference between old and new position in window
NewRelWindowPositionRE := mNewTrackingPosition MOD WindowSize;
DeltaWindowPositionRE := UDINT_TO_DINT(NewRelWindowPositionRE) 
						 - UDINT_TO_DINT(OldRelWindowPositionRE);

OldRelWindowPositionFE := WindowTable[WindowIndexFE].TU_FrontEdgePosition MOD WindowSize;

// Calculate relative TU position in new window
NewRelWindowPositionFE := UDINT_TO_DINT(OldRelWindowPositionFE) + DeltaWindowPositionRE;

// When new position in window is more than one window -> one window can be removed
IF NewRelWindowPositionFE >= WindowSize THEN
	NewWindowIndexFE := WindowIndexFE + 1;
	
	IF NewWindowIndexFE > MaxWindowIndex THEN
		NewWindowIndexFE := NewWindowIndexFE - MaxWindowIndex;
	END_IF
	
	// Copy window
	WindowTable[NewWindowIndexFE] := WindowTable[WindowIndexFE];
	
	ZoneTable[ZoneIndex].TU_StartWindowIndex := NewWindowIndexFE;
	
	// If old window was start of zone, clear window, otherwise mark as reserved 
	// because it is still part of the zone but not of the TU anymore
	IF WindowIndexFE = ZoneTable[ZoneIndex].ZoneStartWindowIndex THEN
		// Clear window
		M_ClearWindow(WindowIndexFE);
		
		ZoneTable[ZoneIndex].ZoneStartWindowIndex := NewWindowIndexFE;
	ELSE
		WindowTable[WindowIndexFE].TU_FrontEdgePosition := 0;
		WindowTable[WindowIndexFE].State := E_WindowTrackingWindowState.RESERVED;
	END_IF
	
// When new position in window is less than 0 -> additional window required
ELSIF NewRelWindowPositionFE < 0 THEN	
	NewWindowIndexFE := WindowIndexFE - 1;
		
	IF NewWindowIndexFE <= 0 THEN
		NewWindowIndexFE := NewWindowIndexFE + MaxWindowIndex;
	END_IF
	
	MovePossible := TRUE;

	// Check if this window consists already of a zone
	IF WindowTable[NewWindowIndexFE].ZoneIndex > 0 THEN
		IF WindowTable[NewWindowIndexFE].ZoneIndex <> ZoneIndex THEN
			// A new window is required which was not part of this zone before (No window with reservation state)
		   UpdateZoneStartWindowIndex := TRUE;

			MovePossible := M_MakeSpace(
								mStartWindowIndex 	:= NewWindowIndexFE,
								mWindowsToFree 		:= 1,
								mAllowZoneDelete 	:= mDeleteTargetZones);
		END_IF
	ELSE
		// A new window is required which was not part of this zone before (No window with reservation state)
		UpdateZoneStartWindowIndex := TRUE;
	END_IF
	
	// If zone of new needed window can not be moved, edge can not be adjusted
	IF NOT MovePossible THEN
		// Move not possible, adjustment failed
		M_AdjustRE := FALSE;
		RETURN;
	END_IF
	
	// If a new window was required to be allocated, update end window index
	IF UpdateZoneStartWindowIndex THEN
		ZoneTable[ZoneIndex].ZoneStartWindowIndex := NewWindowIndexFE;
	END_IF 
	
	// Copy window
	WindowTable[NewWindowIndexFE] := WindowTable[WindowIndexFE];
	
	ZoneTable[ZoneIndex].TU_StartWindowIndex := NewWindowIndexFE;
	
	// Clear exiting rear edge window
	M_ClearWindow(WindowIndexFE);
	
	// Assign window between occupied and takeover same flags
	WindowTable[WindowIndexFE].State := E_WindowTrackingWindowState.OCCUPIED;
	WindowTable[WindowIndexFE].ZoneIndex := ZoneIndex;
	WindowTable[WindowIndexFE].Flush := ZoneTable[ZoneIndex].Flush;

// Window index stays the same
ELSE
	NewWindowIndexFE := WindowIndexFE;
END_IF 

// Correct rear edge and update window and zone
NewAbsWindowPositionFE := DINT_TO_UDINT(NewRelWindowPositionFE) MOD WindowSize + 
					  	  (NewWindowIndexFE -1)*WindowSize;

WindowTable[NewWindowIndexFE].TU_FrontEdgePosition := NewAbsWindowPositionFE;

// If front edge window is first in zone, check position inside window
IF NewWindowIndexFE = ZoneTable[ZoneIndex].ZoneStartWindowIndex THEN
	// Check if adjustment of TU front edge would enlarge zone
	IF ZoneTable[ZoneIndex].ZoneStartPosition > WindowTable[NewWindowIndexFE].TU_FrontEdgePosition THEN
		// Adjust zone start
		// REMARK: Reduce the length OF zone is NOT allowed, because THIS could have influence TO 
    	// minimum gaps between zones
		ZoneTable[ZoneIndex].ZoneStartPosition := WindowTable[NewWindowIndexFE].TU_FrontEdgePosition;
	END_IF
END_IF

// Calculate new length
IF ZoneTable[ZoneIndex].ZoneEndPosition >= ZoneTable[ZoneIndex].ZoneStartPosition THEN
	ZoneTable[ZoneIndex].ZoneLength := UDINT_TO_UINT(ZoneTable[ZoneIndex].ZoneEndPosition 
															   - ZoneTable[ZoneIndex].ZoneStartPosition);
ELSE
	ZoneTable[ZoneIndex].ZoneLength := UDINT_TO_UINT(ZoneTable[ZoneIndex].ZoneEndPosition 
															  + TotalTrackingLength 
															  - ZoneTable[ZoneIndex].ZoneStartPosition);
END_IF

M_AdjustRE := TRUE;
END_METHOD

/// Allocates a fixed zone (Can not be shifted)
/// at a specific position. Position needs to be free. 
METHOD M_AllocateFixedZone : UINT; // > 0 Allocated successfully, otherwise 0
VAR_INPUT
	mActionId				: INT; (* ID of action requests zone - 
								     (0 = Only allocation, but free to be used by other actions) *)
	mAbsolutePosition		: UDINT; // Absolute position on tracking [mm]
	mLength					: UINT; // Length of Zone to be allocated [mm]
	miActionListener		: I_TrackingActionListener; // Action listener of the created zone
	mPositionToLive			: UDINT; // Absolute position until allocation gets deleted automatically if not used (0 = disabled)
END_VAR
VAR
	mStartWindowIndex		: UINT; // Start window index at position
	mTrackingPosition		: UDINT; // Absolute position on tracking
END_VAR
M_AllocateFixedZone := 0;

// Validate inputs
IF mLength <= 0 THEN
	RETURN;
END_IF

// Get window index of absolute position
mStartWindowIndex := M_GetWindowIndex(mAbsolutePosition);

// When a possible location was found
IF mStartWindowIndex > 0 THEN
	mTrackingPosition := M_GetTrackingPosition(mAbsolutePosition);	

	// Allocate zone
	M_AllocateFixedZone := M_ReserveZone(
								mActionId 				:= mActionId,
								mLength					:= mLength, 
								mStartWindowIndex		:= mStartWindowIndex,
								mStartTrackingPosition 	:= mTrackingPosition,
								mInhibitShifting 		:= TRUE,
								miActionListener 		:= miActionListener,
								mPositionToLive 		:= mPositionToLive);				
END_IF
END_METHOD

/// Looks from position ascending for enough space to allocate a new Zone.
METHOD M_AllocateNextFreeZone : UINT; // >0 Index of allocated zone, otherwise 0
VAR_INPUT
	mActionId						: INT; (* ID of action which requests zone - 
								     		(0 = Only allocation, but free to be used by other actions) *)
	mAbsolutePosition				: UDINT; // Absolute position on tracking [mm]
	mLength							: UINT; // Length of Zone to be allocated [mm]
	mMaxDistance					: UDINT; (* Max distance in which begin of a zone is allowed to be allocated (0=Complete distance) 
												Remark: Multiple of windowsize *)
	miActionListener				: I_TrackingActionListener; // Action listener of the created zone
	mPositionToLive					: UDINT; // Absolute position until allocation gets deleted automatically if not used (0 = disabled)
END_VAR
VAR
	mStartWindowIndex				: UINT; // Start Window index to search for enough space
	mNumberLengthWindows			: UINT; // Lenght represented as windows
	RemainingWindowLength 			: INT; // Remaining length on tracking, before reaching startpoint [windows]
	mWindowsTrackingEnd 			: UDINT; // Number of windows from a requesting position to the end of tracking length 
	mWindowIndex 					: UINT; // Iterating window index
	mCounterFreeWindows 			: UINT; // Counter of free windows in a row
	mFreeStartWindowIndex 			: UINT; // Found start window index
	mFreeStartTrackingPosition		: UDINT; // Position in start window index
	mIdx							: DINT; // Loop iterator
	mTrackingPosition				: UDINT; // Absolute position on tracking
	mRelWindowPositionZoneStart		: UDINT; // Relative window position of zone start
	mFullLength						: UINT; // Full required length for allocation
	mMaxDistanceWindows				: INT; // Max windows to be checked if distance is limited
END_VAR
M_AllocateNextFreeZone := 0;

// Get window index of absolute position
mStartWindowIndex := M_GetWindowIndex(mAbsolutePosition);
mTrackingPosition := M_GetTrackingPosition(mAbsolutePosition);	

// Validate inputs
IF mLength <= 0 OR 
   mStartWindowIndex = 0 THEN
	RETURN;
END_IF

// Convert length into number of windows
IF WindowSize > 0 THEN
	// Calculate relative position in first zone window
	mRelWindowPositionZoneStart := mTrackingPosition MOD WindowSize;
	
	// The relative position in the first window is added to the length, 
	// in order to get the amount of windows which are allocated for that TU finally
	mFullLength := mLength + UDINT_TO_UINT(mRelWindowPositionZoneStart);
	
	// Convert length into number of windows
	mNumberLengthWindows := mFullLength / WindowSize;
	// If not the full length could be mapped in windows
	// add an additional window
	IF (mFullLength MOD WindowSize) > 0 THEN
		mNumberLengthWindows := mNumberLengthWindows + 1;
	END_IF
ELSE
	// Error
	mNumberLengthWindows := 0;
	RETURN;
END_IF

// When zones get deleted on tracking end, the valid tracking distance for allocaition
// is limited to the windows up to the absolute positions and the trackinglength backwards.
// Therefore from the whole distance all windows of TrackingLength - AbsolutePosition have
// to be removed from the allowed shifting distance.
IF DeleteZoneTrackingEnd THEN
	IF WindowSize > 0 THEN
		mWindowsTrackingEnd := (TrackingLength - mAbsolutePosition) / WindowSize + 1;	
	ELSE
		// Configuration error
		mWindowsTrackingEnd := 0;
	END_IF
	
	RemainingWindowLength := UINT_TO_INT(MaxWindowIndex) - UDINT_TO_INT(mWindowsTrackingEnd) - 1;
ELSE
	RemainingWindowLength := UINT_TO_INT(MaxWindowIndex) - 1;
END_IF
	
// When no limitations are given for allocation
IF mMaxDistance = 0 THEN
	mMaxDistanceWindows := UINT_TO_INT(MaxWindowIndex);
// Otherwise limit windows to be checked
ELSE
	// Convert length into number of windows
	mMaxDistanceWindows := UDINT_TO_INT(mMaxDistance / WindowSize);
	// If not the full length could be mapped in windows
	// add an additional window
	IF (mMaxDistance MOD WindowSize) > 0 THEN
		mMaxDistanceWindows := mMaxDistanceWindows + 1;
	END_IF
END_IF

mWindowIndex := mStartWindowIndex;
mFreeStartTrackingPosition := mTrackingPosition;
mCounterFreeWindows := 0;

// Search ascending for enough window space
FOR mIdx := 1 TO WindowTracking.MAX_NUMBER_OF_WINDOWS DO
	// No space available for allocaiton, request failed
	IF RemainingWindowLength <= 0 THEN
		mFreeStartWindowIndex := 0;
		M_AllocateNextFreeZone := 0;
		EXIT;
		
	// Max distance expired and still no zone found
	ELSIF mMaxDistanceWindows <= 0 AND 
          mCounterFreeWindows = 0 THEN
		mFreeStartWindowIndex := 0;
		M_AllocateNextFreeZone := 0;
		EXIT;
		
	// When window is not attached to a zone and not
	// marked to be flushed, its a valid free window
	ELSIF WindowTable[mWindowIndex].ZoneIndex = 0 AND 
       NOT WindowTable[mWindowIndex].Flush THEN
	   
	    IF mCounterFreeWindows = 0 THEN
			// If start window is different than found window index, 
			// set to begin of zone
			IF mWindowIndex <> mStartWindowIndex THEN 
				mFreeStartTrackingPosition := (mWindowIndex - 1) * WindowSize;
			END_IF
			
			mFreeStartWindowIndex := mWindowIndex;
		END_IF
		
		mCounterFreeWindows := mCounterFreeWindows + 1;
		
		// When enough free windows are found, 
		// leave loop to allocate 
		IF mCounterFreeWindows >= mNumberLengthWindows THEN
			EXIT;
		END_IF
	ELSE
		// Reset counter and startposition of free windows in a row
		mCounterFreeWindows := 0;
		mFreeStartWindowIndex := 0;
	END_IF
	
	mWindowIndex := mWindowIndex + 1;
	
	// Correct window border overflow
	IF mWindowIndex > MaxWindowIndex THEN
		mWindowIndex := mWindowIndex - MaxWindowIndex;
	END_IF
	
	// Calculate remaining possible windows wich can be used
	// for allocation
	RemainingWindowLength := RemainingWindowLength - 1;
	
	// Decrease amount of windows in which a zone needs to found for allocation
	mMaxDistanceWindows := mMaxDistanceWindows - 1;
END_FOR

// When a possible location was found
IF mFreeStartWindowIndex > 0 THEN
	// Allocate zone
	M_AllocateNextFreeZone := M_ReserveZone(
								mActionId 				:= mActionId,
								mLength					:= mLength, 
								mStartWindowIndex 		:= mFreeStartWindowIndex,
								mStartTrackingPosition 	:= mFreeStartTrackingPosition,
								mInhibitShifting 		:= FALSE,
								miActionListener 		:= miActionListener,
								mPositionToLive 		:= mPositionToLive);
END_IF
END_METHOD

// Assigns an already allocated but free zone, beginning at absolute position upstream
// Remark: No zones are allocated, only existing zones are considered.
METHOD M_AssignNextFreeZone : UINT // Returns index of assigned zone if successful, otherwise 0
VAR_INPUT
	mActionId				: INT; // ID of action which requests zone (<>0)
	mAbsolutePosition		: UDINT; // Absolute Start position on the tracking [mm]
	mMaxDistance			: UDINT; // Max distance in which begin of a zone is allowed to be for assignment (0=Complete distance) 
	mLength					: UINT; // Length of Zone to be allocated [mm]
	miActionListener		: I_TrackingActionListener; // Action listener of the created zone
	mPositionToLive			: UDINT; // Absolute position until allocation gets deleted automatically if not used (0 = disabled)
END_VAR
VAR
	mIdx					: UINT; // Loop iterator
	mZoneIndex				: UINT; // Zone index
	mZoneCounter 			: INT; // Amount of already considerd zones
	mFoundZoneIndex			: UINT; // Possible zone index
	mDistanceToLastFoundZone: UDINT; // Distance from Abspoint to last found zone
	mDistanceToCurrentZone	: UDINT; // Distance from abspoint to current found zone
	mMaxAssignDistance		: UDINT; // Max distance which is covered to assign a zone
	mTrackingPosition		: UDINT; // Abs position on tracking
END_VAR
M_AssignNextFreeZone := 0;
mZoneIndex := 0;

// Validate inputs
IF mLength <= 0 OR
   mActionId = 0 THEN
	RETURN;
END_IF

// Abort if no zones available at all
IF ZoneCount = 0 THEN
	RETURN;
END_IF

IF mMaxDistance = 0 THEN	
	mMaxAssignDistance := TotalTrackingLength;
ELSE
	mMaxAssignDistance := mMaxDistance;
END_IF

// Translate requesting position into tracking position
mTrackingPosition := M_GetTrackingPosition(mAbsolutePosition);

mZoneCounter := 0;
mFoundZoneIndex := 0;
mDistanceToLastFoundZone := TotalTrackingLength;

// Check all allocated zones to determine the nearest possible to AbsPosition
// Remark: As a reason of performance no scan through all windows upstream is initiated.
FOR mIdx := 1 TO WindowTracking.MAX_NUMBER_OF_ZONES DO
	// When all zones are considered, stop
	IF mZoneCounter = ZoneCount THEN
		EXIT;
		
